(* CODESYS project Tc3_Component.library
   Description: State Model with Observer and Events
   Author: Peter Zerlauth
   Company: Zerlauth
   Version: 0.0.0.1
   Title: Tc3_Component
   DefaultNamespace: Tc3_Component
   Placeholder: Tc3_Component

Project tree, tasks and I/O mapping:
  libraries: Tc2_Standard, * (Beckhoff Automation GmbH); Tc2_System, * (Beckhoff Automation GmbH); Tc2_Utilities, * (Beckhoff Automation GmbH); Tc3_JsonXml, * (Beckhoff Automation GmbH)
  Component/
    Event/
      Observable/
        function block FB_Observable [ST]: FB_exit, M_Attach, M_Clear, M_Detach, M_Find, M_Index, M_Notify, P_Length
        interface I_Observable: M_Attach, M_Detach, P_Length
        interface I_Observer: M_Notify
      data type E_Event
      function block FB_Event [ST]: FB_init, M_Abort, M_AddBOOL, M_AddINT, M_AddREAL, M_AddSTRING, M_AddTIME, M_Arguments, M_Debug, M_Default, M_Error, M_Info, M_Stop, M_Warning, P_History, P_Logger, P_Observer
      interface I_Event: M_Abort, M_AddBOOL, M_AddINT, M_AddREAL, M_AddSTRING, M_AddTIME, M_Debug, M_Error, M_Info, M_Stop, M_Warning, P_History, P_Logger, P_Observer
      data type ST_Event
      data type ST_EventFlags
    Info/
      function block FB_Info [ST]: M_Initialise, P_Class, P_Comment, P_ID, P_Instance, P_Timestamp
      interface I_Info: P_Class, P_Comment, P_ID, P_Instance, P_Timestamp
    Sequence/
      data type E_Sequence
      function block FB_Sequence [ST]: FB_init, M_Await, M_Reset, M_Restore, M_Save, M_Set, P_History, P_Message, P_Number
      interface I_Sequence: M_Await, M_Reset, M_Set, P_History, P_Message, P_Number
      data type ST_Sequence
    data type E_RequestMode
    data type E_RequestState
    data type E_State
    function block FB_Component [ST]: M_RequestMode, M_RequestState, M_Aborted, M_Aborting, M_Completed, M_Completing, M_Execute, M_Held, M_Holding, M_Idle, M_Initialise, M_Paused, M_Pausing, M_Resetting, M_Resuming, M_Running, M_Starting, M_Stopped, M_Stopping, M_Unholding, FB_init, M_Cycle, M_Notify, M_OnMode, M_OnState, P_Event, P_Info, P_Mode, P_Sequence, P_State
    interface I_Component: M_Cycle, M_RequestMode, M_RequestState, P_Event, P_Info, P_Mode, P_State
    interface I_Cycle: M_Cycle
  Function/
    function block FB_Function [ST]
  Images/
    StateModel.svg
    test.jpg
  00000000-0000-0000-0000-000000000000|Images\StateModel.svg
  00000000-0000-0000-0000-000000000000|Images\test.jpg
  Layers/
    Layer/
      function block FB_Layer [ST]: M_Attach, M_Dettach, M_Notify, M_Resetting, M_Starting, P_Delay, P_List, P_Next, P_Timeout
      interface I_Layer: M_Attach, M_Dettach, P_Delay, P_List, P_Next, P_Timeout
    function block FB_Layers [ST]: M_Cycle, P_E0, P_E1, P_On
    interface I_Layers: P_E0, P_E1, P_On
  List/
    function block FB_ListComponent [ST]: FB_exit, M_Add, M_Clear, M_Find, M_Index, M_Remove, P_Length
    function block FB_ListObject [ST]: FB_exit, M_Add, M_Clear, M_Find, M_Index, M_Remove, P_Length
    function block FB_ListString [ST]: FB_exit, M_Add, M_Clear, M_Find, M_Index, M_Remove, P_Length
    interface I_ListBase: M_Clear, P_Length
    interface I_ListComponent: M_Add, M_Find, M_Index, M_Remove
    interface I_ListObject: M_Add, M_Find, M_Index, M_Remove
    interface I_ListString: M_Add, M_Find, M_Index, M_Remove
  Logger/
    function block FB_AbstractLogger [ST]: M_Log, P_LogLevel
    function block FB_GlobalLogger [ST]: M_Find, M_Log
    function block FB_ListObject_1 [ST]: FB_exit, M_Add, M_Clear, M_Find, M_Index, M_Remove, P_Length
    function block FB_Logger [ST]: M_Delete, M_Find, M_Log, M_Reset, P_Events, P_Length
    function block FB_TcLogger [ST]: M_Find, M_Log, M_Reset
    interface I_Logger: M_Log
  Module/
    function block FB_Module [ST]: M_Aborted, M_Completing, M_Cycle, M_Holding, M_Idle, M_Initialise, M_OnMode, M_Pausing, M_Resetting, M_Resuming, M_Running, M_Starting, M_Stopped, M_Unholding, P_Layers
    interface I_Module: P_Layers
  Object/
    function block FB_Object [ST]
    interface I_Object
  Utils/
    Analog/
      function block AnalogInput [ST]: P_ID, P_State, P_Value
      function block AnalogInputREAL [ST]: P_ID, P_State, P_Value
      function block AnalogOutput [ST]: FB_init, P_ID, P_State, P_Value
      interface I_AnalogChannel: P_Value
    Digital/
      function block FB_DigitalInput [ST]: P_ID, P_State, P_Value
      function block FB_DigitalOutput [ST]: P_ID, P_State, P_Value
      interface I_Channel: P_ID, P_State
      interface I_DigitalChannel: P_Value
    File/
      function block FB_File [ST]: M_Append, M_AppendLine, M_Close, M_Create, M_Delete, M_Load, M_Open, M_Read, M_Write, P_Error
      interface I_File: M_Append, M_AppendLine, M_Close, M_Create, M_Delete, M_Load, M_Open, M_Read, M_Write, P_Error
    function block FB_ArrayDint [ST]
    function block FB_Debounce [ST]: P_Value
  Version/
    global variables Global_Version
  global variables Globals
  global variables Parameters
*)

// Component/Event/E_Event
{attribute 'qualified_only'}
{attribute 'strict'}
{attribute 'to_string'}
TYPE E_Event :
(
	Verbose			:= 0,
	Debug			:= 1,
	Information		:= 2,
	Warning			:= 3,
	Error			:= 4
);
END_TYPE

// Component/Event/ST_Event
{attribute 'analysis' := '-33'}
TYPE ST_Event :
	STRUCT
		iSource:		I_Component;
		eEventType:		E_Event;
		nTimestamp:   	ULINT;
		nID:			ULINT;
		sInstance:		STRING(255);
		sClass:			STRING(255);
		sMessage:		STRING(255);
		sDefault:		STRING(255);
		sArguments:		STRING(255);
		stFlags:		ST_EventFlags;
	END_STRUCT
END_TYPE

// Component/Event/ST_EventFlags
{attribute 'analysis' := '-33'}
TYPE ST_EventFlags :
STRUCT
	bActive:		BIT;
	bRemove:		BIT;
END_STRUCT
END_TYPE

// Component/Sequence/E_Sequence
{attribute 'qualified_only'}
{attribute 'strict'}
{attribute 'to_string'}

TYPE E_Sequence :
(
	Manual			:= -32768,
	{attribute 'analysis' := '-27'}
	Start			:= 0,
	Done			:= 32767
);
END_TYPE

// Component/Sequence/ST_Sequence
TYPE ST_Sequence :
STRUCT
	sMessage:				STRING(255);
	nNumber:				INT;
END_STRUCT
END_TYPE

// Component/E_RequestMode
{attribute 'qualified_only'}
{attribute 'strict'}
{attribute 'to_string'}
TYPE E_RequestMode :
(
	{attribute 'hide'}
    Undefined   := 0,
	Automatic   := 1,
    Semiauto    := 2,
	Manual		:= 3
);
END_TYPE

// Component/E_RequestState
{attribute 'qualified_only'}
{attribute 'strict'}
{attribute 'to_string'}

TYPE E_RequestState :
(
	{attribute 'hide'}
    Undefined   := 0,
	{attribute 'analysis' := '-27'}
	Reset       := 1,
	{attribute 'analysis' := '-27'}
    Start       := 2,
    Pause       := 4,	
    Hold      	:= 8,
	Complete	:= 16,	
	Stop		:= 32,
	Abort       := 64
);
END_TYPE

// Component/E_State
{attribute 'qualified_only'}
{attribute 'strict'}
{attribute 'to_string'}
TYPE E_State :
(
	{attribute 'hide'}
	Undefined		:= 0,
	Idle			:= 1,
	
// Start
	Starting		:= 2,
	Execute			:= 3,
	
// Pause
	Pausing			:= 4,
	Paused			:= 5,
	Resuming		:= 6,
	
// Hold
	Holding			:= 7,
	Held			:= 8,
	Unholding		:= 9,
	
// Complete
	Completing		:= 10,
	Completed		:= 11,

// Stop
	Stopping		:= 12,
	Stopped			:= 13,

// Abort	
	Aborting		:= 14,
	Aborted			:= 15,

// Reset
	Resetting		:= 16

);
END_TYPE

// Version/Global_Version
{attribute 'TcGenerated'}
{attribute 'no-analysis'}
{attribute 'linkalways'}
// This function has been automatically generated from the project information.
VAR_GLOBAL CONSTANT
	{attribute 'const_non_replaced'}
	stLibVersion_Tc3_Component : ST_LibVersion := (iMajor := 0, iMinor := 0, iBuild := 0, iRevision := 1, nFlags := 0, sVersion := '0.0.0.1');
END_VAR

// Globals
VAR_GLOBAL
	{IF (defined (release))}
    	{attribute 'hide'}
	{END_IF}
	fbLogger:			FB_GlobalLogger;		// Global Logger, as default without module
	{attribute 'analysis' := '-33'}
	bSimulation:		BOOL;
END_VAR

// Parameters
{attribute 'qualified_only'}
VAR_GLOBAL CONSTANT
	{attribute 'analysis' := '-33'}
	nSequence:						UINT:= 9;		// Maximum of Sequence history
	{attribute 'analysis' := '-33'}
	nList:							UINT:= 46;		// Maximum of displayed items in list
END_VAR

// Component/Event/Observable/FB_Observable
{attribute 'no_explicit_call'} 
FUNCTION_BLOCK PUBLIC FB_Observable IMPLEMENTS I_Observable
VAR_INPUT
	iParent:		I_Component;	
END_VAR
VAR
	pList: 			POINTER TO I_Component;
    {attribute 'hide'}
	nLength:		DINT;
	{IF (defined (release))}
    	{attribute 'hide'}
	{END_IF}
	aList:			POINTER TO POINTER TO ARRAY [0..100] OF I_Component:=ADR(pList);
END_VAR

// https://github.com/PeterZerlauth/Tc3_Component

METHOD FB_exit : BOOL
VAR_INPUT
	bInCopyCode : BOOL; // if TRUE, the exit method is called for exiting an instance that is copied afterwards (online change).
END_VAR
M_Clear();
END_METHOD

METHOD M_Attach : BOOL
VAR_INPUT
	Object: 	I_Component;
END_VAR
VAR
	pOldList: 	POINTER TO I_Component;
END_VAR
IF Object <> 0 THEN
	// First Item
	IF pList = 0 THEN
		nLength:= nLength + 1;
		pList:= __NEW(POINTER TO I_Component,DINT_TO_UDINT(nLength));
	ELSE
		// Item already in List
		IF M_Find(Object) = -1 THEN
			// backup 
			pOldList:= pList;
			// new Length
			nLength:= nLength + 1;
			// new pointer
			pList:= __NEW(POINTER TO I_Component,DINT_TO_UDINT(nLength));
			// restore
			Memcpy(pList,pOldList, SIZEOF(POINTER TO I_Component)*DINT_TO_UDINT(nLength -1));
			// delete old
			__DELETE(pOldList);
		ELSE
			M_Attach:= FALSE;	
			RETURN;
		END_IF
	END_IF
	IF pList = 0 THEN
		RETURN;
	END_IF
	// add new Object
	pList[nLength-1]:= Object;
	M_Attach:= TRUE;
ELSE
	M_Attach:= FALSE;	
END_IF
END_METHOD

METHOD M_Clear
IF pList <> 0 THEN
	nLength:= 0;
	__DELETE(pList);
END_IF
END_METHOD

METHOD M_Detach : BOOL
VAR_INPUT
	Object: 	I_Component;
END_VAR
VAR
	pOldList:			POINTER TO I_Component;
	nPosition: 			DINT;
END_VAR
IF Object <> 0 THEN
	// First Item
	IF nLength >= 0 THEN
		// Item already in List
		nPosition:= M_Find(Object);
		IF nPosition <> -1 THEN
			// backup 
			pOldList:= pList;
			// new Length
			nLength:= nLength -1;
			// new pointer
			pList:= __NEW(POINTER TO I_Component,DINT_TO_UDINT(nLength));
			// restore lower part
			Memcpy(pList,pOldList, SIZEOF(POINTER TO I_Component) * DINT_TO_UDINT(nPosition));
			//pList[nPosition]:= iObject;
			Memcpy(pList + (SIZEOF(POINTER TO I_Component)*nPosition),pOldList + (SIZEOF(POINTER TO I_Component)*(nPosition + 1)), SIZEOF(POINTER TO I_Component) * DINT_TO_UDINT(nLength - nPosition));
			// delete old
			__DELETE(pOldList);
		ELSE
			M_Detach:= FALSE;	
			RETURN;
		END_IF
	ELSE
		M_Detach:= FALSE;	
		RETURN;
	END_IF
	M_Detach:= TRUE;
ELSE
	M_Detach:= FALSE;	
END_IF
END_METHOD

METHOD M_Find : DINT
VAR_INPUT
	Object: 	I_Component;
END_VAR
VAR
	nIndex: 	UINT;
END_VAR
// Object already in List
M_Find := -1;
WHILE nIndex < nLength DO
    IF (pList[nIndex] = Object) THEN
        M_Find := nIndex;
        RETURN;
    END_IF
	nIndex := nIndex + 1;
END_WHILE
END_METHOD

METHOD M_Index : I_Observer
VAR_INPUT
	Index: 	DINT;
END_VAR
IF Index <= nLength THEN
	M_Index:= pList[Index];
END_IF
END_METHOD

METHOD M_Notify
VAR_INPUT
	iSender:		I_Component;
	eRequest:		E_RequestState;
END_VAR

VAR
	nIndex: 		DINT;
END_VAR
// Prevent Infinite loop from callbacks
WHILE nIndex < nLength DO
	IF pList[nIndex] <> iSender THEN
		pList[nIndex].M_Notify(iParent, eRequest);		
	END_IF
	nIndex:= nIndex + 1; 
END_WHILE
END_METHOD

{attribute 'OPC.UA.DA.Property' := '1'}
{attribute 'monitoring' := 'call'}
PROPERTY P_Length : DINT
GET
P_Length:= nLength;
END_GET
END_PROPERTY

END_FUNCTION_BLOCK

// Component/Event/Observable/I_Observable
INTERFACE I_Observable EXTENDS I_Observer

METHOD PUBLIC M_Attach : BOOL
VAR_INPUT
	Object: 	I_Component;
END_VAR
END_METHOD

METHOD PUBLIC M_Detach : BOOL
VAR_INPUT
	Object: 	I_Component;
END_VAR
END_METHOD

{attribute 'OPC.UA.DA.Property' := '1'}
{attribute 'monitoring' := 'call'}
PROPERTY P_Length : DINT
GET
END_GET
END_PROPERTY

END_INTERFACE

// Component/Event/Observable/I_Observer
INTERFACE I_Observer EXTENDS I_Object

METHOD PUBLIC M_Notify
VAR_INPUT
	iSender:		I_Component;
	eRequest:		E_RequestState;
END_VAR
END_METHOD

END_INTERFACE

// Object/I_Object
INTERFACE I_Object EXTENDS __SYSTEM.IQueryInterface

END_INTERFACE

// Component/I_Component
INTERFACE I_Component EXTENDS I_Observer, I_Cycle

METHOD PUBLIC M_Cycle
VAR_INPUT
END_VAR
END_METHOD

METHOD PUBLIC M_RequestMode : BOOL
VAR_INPUT
	eMode:		E_RequestMode;
END_VAR
END_METHOD

METHOD PUBLIC M_RequestState : BOOL
VAR_INPUT
	eRequest:	E_RequestState;
END_VAR
END_METHOD

PROPERTY PUBLIC P_Event : I_Event
GET
END_GET
END_PROPERTY

{attribute 'OPC.UA.DA.Property' := '1'}
{attribute 'monitoring' := 'call'}
PROPERTY PUBLIC P_Info : I_Info
GET
END_GET
END_PROPERTY

{attribute 'OPC.UA.DA.Property' := '1'}
{attribute 'monitoring' := 'call'}
PROPERTY PUBLIC P_Mode : E_RequestMode
GET
END_GET
END_PROPERTY

{attribute 'OPC.UA.DA.Property' := '1'}
{attribute 'monitoring' := 'call'}
PROPERTY PUBLIC P_State : E_State
GET
END_GET
END_PROPERTY

END_INTERFACE

// Component/I_Cycle
INTERFACE I_Cycle EXTENDS I_Object

METHOD PUBLIC M_Cycle
VAR_INPUT
END_VAR
END_METHOD

END_INTERFACE

// Component/Event/I_Event
INTERFACE I_Event EXTENDS I_Object

METHOD PUBLIC M_Abort
VAR_INPUT
	sMessage:				STRING(255);
	nID:					ULINT;
END_VAR
END_METHOD

METHOD PUBLIC M_AddBOOL : I_Event
VAR_INPUT
	Value: 	BOOL;
END_VAR
END_METHOD

METHOD PUBLIC M_AddINT : I_Event
VAR_INPUT
	Value: 	LINT;
END_VAR
END_METHOD

METHOD PUBLIC M_AddREAL : I_Event
VAR_INPUT
	Value: 	Lreal;
	Decimals: INT;
END_VAR
END_METHOD

METHOD PUBLIC M_AddSTRING : I_Event
VAR_INPUT
	Value: STRING(255);
END_VAR
END_METHOD

METHOD PUBLIC M_AddTIME : I_Event
VAR_INPUT
	Value: 	TIME;
END_VAR
END_METHOD

METHOD PUBLIC M_Debug
VAR_INPUT
	sMessage:				STRING(255);
END_VAR
END_METHOD

METHOD PUBLIC M_Error
VAR_INPUT
	sMessage:				STRING(255);
	nID:					ULINT;
END_VAR
END_METHOD

METHOD PUBLIC M_Info
VAR_INPUT
	sMessage:				STRING(255);
	nID:					ULINT;
END_VAR
END_METHOD

METHOD PUBLIC M_Stop
VAR_INPUT
	sMessage:				STRING(255);
	nID:					ULINT;
END_VAR
END_METHOD

METHOD PUBLIC M_Warning
VAR_INPUT
	sMessage:				STRING(255);
	nID:					ULINT;
END_VAR
END_METHOD

{attribute 'OPC.UA.DA.Property' := '1'}
{attribute 'monitoring' := 'call'}
{attribute 'suppress_wrn_C0410'}
PROPERTY PUBLIC P_History : REFERENCE TO ARRAY [0..5] OF ST_Event;
GET
END_GET
SET
END_SET
END_PROPERTY

PROPERTY PUBLIC P_Logger : I_Logger
GET
END_GET
SET
END_SET
END_PROPERTY

PROPERTY PUBLIC P_Observer : I_Observable
GET
END_GET
END_PROPERTY

END_INTERFACE

// Logger/I_Logger
INTERFACE I_Logger EXTENDS I_Object

METHOD PUBLIC M_Log
VAR_INPUT
	{attribute 'analysis' := '-33'}
	stEvent	: ST_Event;
END_VAR
END_METHOD

END_INTERFACE

// Component/Info/I_Info
INTERFACE I_Info EXTENDS I_Object

{attribute 'OPC.UA.DA.Property' := '1'}
{attribute 'monitoring' := 'call'}
PROPERTY PUBLIC P_Class : STRING(255)
GET
END_GET
END_PROPERTY

{attribute 'OPC.UA.DA.Property' := '1'}
{attribute 'monitoring' := 'call'}
PROPERTY PUBLIC P_Comment : STRING(255)
GET
END_GET
END_PROPERTY

{attribute 'OPC.UA.DA.Property' := '1'}
{attribute 'monitoring' := 'call'}
PROPERTY PUBLIC P_ID : STRING(25)
GET
END_GET
SET
END_SET
END_PROPERTY

{attribute 'OPC.UA.DA.Property' := '1'}
{attribute 'monitoring' := 'call'}
PROPERTY PUBLIC P_Instance : STRING(255)
GET
END_GET
END_PROPERTY

{attribute 'OPC.UA.DA.Property' := '1'}
{attribute 'monitoring' := 'call'}
PROPERTY PUBLIC P_Timestamp : ULINT
GET
END_GET
END_PROPERTY

END_INTERFACE

// Component/Event/FB_Event
FUNCTION_BLOCK FB_Event IMPLEMENTS I_Event
VAR_INPUT
	fbObserver:			FB_Observable;				// Observer
END_VAR
VAR_OUTPUT
END_VAR
VAR
	iLogger:			I_Logger;
	iParent:			I_Component;				// Parent component
    {attribute 'hide'}
	fbList:				FB_ListString;				// contains a list with string values

	stEvent:			ST_Event;					// Event
    {attribute 'hide'}
	aHistory:			ARRAY [0..5] OF ST_Event;	// History of events
END_VAR

// https://github.com/PeterZerlauth/Tc3_Component

METHOD FB_init : BOOL
VAR_INPUT
	bInitRetains : BOOL; // if TRUE, the retain variables are initialized (warm start / cold start)
	bInCopyCode : BOOL;  // if TRUE, the instance afterwards gets moved into the copy code (online change)
	iParent:			I_Component;
END_VAR
THIS^.iParent:= iParent;
fbObserver.iParent:= iParent;
END_METHOD

METHOD PUBLIC M_Abort
VAR_INPUT
	sMessage:				STRING(255);
	nID:					ULINT;
END_VAR
stEvent.sMessage:= sMessage;
stEvent.iSource:= iParent;
stEvent.sInstance:= iParent.P_Info.P_Instance;
stEvent.sClass:= iParent.P_Info.P_Class;
stEvent.eEventType:= E_Event.Error;
stEvent.nTimestamp:= F_GetSystemTime();
stEvent.nID:= nID;
stEvent.sDefault:= M_Default(sMessage);
stEvent.sArguments:= M_Arguments();
stEvent.stFlags.bActive:= TRUE;
stEvent.stFlags.bRemove:= FALSE;

IF iLogger = 0 THEN
	fbLogger.M_Log(stEvent);
ELSE
	iLogger.M_Log(stEvent);
END_IF

iParent.M_RequestState(E_RequestState.Abort);

fbObserver.M_Notify(iParent, E_RequestState.Abort);

IF aHistory[0].sMessage <> stEvent.sMessage THEN
	MemCpy(ADR(aHistory[1]), ADR(aHistory[0]), SIZEOF(ST_Event) * 5);
	aHistory[0]:= stEvent;
END_IF
END_METHOD

METHOD PUBLIC M_AddBOOL : I_Event
VAR_INPUT
	Value: 	bool;
END_VAR
fbList.M_Add(BOOL_TO_STRING(Value));
M_AddBOOL:= THIS^;
END_METHOD

METHOD PUBLIC M_AddINT : I_Event
VAR_INPUT
	Value: 	LINT;
END_VAR
fbList.M_Add(LINT_TO_STRING(Value));
M_AddINT:= THIS^;
END_METHOD

METHOD PUBLIC M_AddREAL : I_Event
VAR_INPUT
	Value: 	Lreal;
	Decimals: INT;
END_VAR
fbList.M_Add(LREAL_TO_FMTSTR(Value, Decimals, TRUE));
M_AddREAL:= THIS^;
END_METHOD

METHOD PUBLIC M_AddSTRING : I_Event
VAR_INPUT
	Value: STRING(255);
END_VAR
fbList.M_Add(Value);
M_AddSTRING:= THIS^;
END_METHOD

METHOD PUBLIC M_AddTIME : I_Event
VAR_INPUT
	Value: 	TIME;
END_VAR
fbList.M_Add(TIME_TO_STRING(Value));
M_AddTIME:= THIS^;
END_METHOD

METHOD INTERNAL M_Arguments : STRING(255)
VAR_INPUT
END_VAR
VAR
	nIndex:			INT;
END_VAR
WHILE nIndex < fbList. P_Length DO
	M_Arguments:= Concat(Concat(M_Arguments, fbList.M_Index(nIndex)), '$N');
	nIndex:= nIndex + 1;
END_WHILE

fbList.M_Clear();
END_METHOD

METHOD PUBLIC M_Debug
VAR_INPUT
	sMessage:				STRING(255);
END_VAR
stEvent.sMessage:= sMessage;
stEvent.iSource:= iParent;
stEvent.sInstance:= iParent.P_Info.P_Instance;
stEvent.sClass:= iParent.P_Info.P_Class;
stEvent.eEventType:= E_Event.Debug;
stEvent.nTimestamp:= F_GetSystemTime();
stEvent.nID:= 0;
stEvent.sDefault:= M_Default(sMessage);
stEvent.sArguments:= M_Arguments();
stEvent.stFlags.bActive:= TRUE;
stEvent.stFlags.bRemove:= TRUE;

IF iLogger = 0 THEN
	fbLogger.M_Log(stEvent);
ELSE
	iLogger.M_Log(stEvent);
END_IF

IF aHistory[0].sMessage <> stEvent.sMessage THEN
	MemCpy(ADR(aHistory[1]), ADR(aHistory[0]), SIZEOF(ST_Event) * 5);
	aHistory[0]:= stEvent;
END_IF
END_METHOD

METHOD INTERNAL M_Default : STRING(255)
VAR_INPUT
	sMessage:		STRING(255);
END_VAR
VAR
	nIndex:		   	DINT;
	nPosition: 		INT;
END_VAR
nPosition:= Find(sMessage, '%s');
WHILE nPosition <> 0 DO
	sMessage:= Replace(sMessage, fbList.M_Index(nIndex), 2, nPosition);
	nPosition:= Find(sMessage, '%s');
	nIndex:= nIndex + 1;
END_WHILE
M_Default:= sMessage;
END_METHOD

METHOD PUBLIC M_Error
VAR_INPUT
	sMessage:				STRING(255);
	nID:					ULINT;
END_VAR
stEvent.sMessage:= sMessage;
stEvent.iSource:= iParent;
stEvent.sInstance:= iParent.P_Info.P_Instance;
stEvent.sClass:= iParent.P_Info.P_Class;
stEvent.eEventType:= E_Event.Error;
stEvent.nTimestamp:= F_GetSystemTime();
stEvent.nID:= nID;
stEvent.sDefault:= M_Default(sMessage);
stEvent.sArguments:= M_Arguments();
stEvent.stFlags.bActive:= TRUE;
stEvent.stFlags.bRemove:= TRUE;

IF iLogger = 0 THEN
	fbLogger.M_Log(stEvent);
ELSE
	iLogger.M_Log(stEvent);
END_IF

IF aHistory[0].sMessage <> stEvent.sMessage THEN
	MemCpy(ADR(aHistory[1]), ADR(aHistory[0]), SIZEOF(ST_Event) * 5);
	aHistory[0]:= stEvent;
END_IF
END_METHOD

METHOD PUBLIC M_Info
VAR_INPUT
	sMessage:				STRING(255);
	nID:					ULINT;
END_VAR
stEvent.sMessage:= sMessage;
stEvent.iSource:= iParent;
stEvent.sInstance:= iParent.P_Info.P_Instance;
stEvent.sClass:= iParent.P_Info.P_Class;
stEvent.eEventType:= E_Event.Information;
stEvent.nTimestamp:= F_GetSystemTime();
stEvent.nID:= nID;
stEvent.sDefault:= M_Default(sMessage);
stEvent.sArguments:= M_Arguments();
stEvent.stFlags.bActive:= TRUE;
stEvent.stFlags.bRemove:= TRUE;

IF iLogger = 0 THEN
	fbLogger.M_Log(stEvent);
ELSE
	iLogger.M_Log(stEvent);
END_IF

IF aHistory[0].sMessage <> stEvent.sMessage THEN
	MemCpy(ADR(aHistory[1]), ADR(aHistory[0]), SIZEOF(ST_Event) * 5);
	aHistory[0]:= stEvent;
END_IF
END_METHOD

METHOD PUBLIC M_Stop
VAR_INPUT
	sMessage:				STRING(255);
	nID:					ULINT;
END_VAR
stEvent.sMessage:= sMessage;
stEvent.iSource:= iParent;
stEvent.sInstance:= iParent.P_Info.P_Instance;
stEvent.sClass:= iParent.P_Info.P_Class;
stEvent.eEventType:= E_Event.Error;
stEvent.nTimestamp:= F_GetSystemTime();
stEvent.nID:= nID;
stEvent.sDefault:= M_Default(sMessage);
stEvent.sArguments:= M_Arguments();
stEvent.stFlags.bActive:= TRUE;
stEvent.stFlags.bRemove:= FALSE;

IF iLogger = 0 THEN
	fbLogger.M_Log(stEvent);
ELSE
	iLogger.M_Log(stEvent);
END_IF

iParent.M_RequestState(E_RequestState.Stop);

fbObserver.M_Notify(iParent, E_RequestState.Abort);

IF aHistory[0].sMessage <> stEvent.sMessage THEN
	MemCpy(ADR(aHistory[1]), ADR(aHistory[0]), SIZEOF(ST_Event) * 5);
	aHistory[0]:= stEvent;
END_IF
END_METHOD

METHOD PUBLIC M_Warning
VAR_INPUT
	sMessage:				STRING(255);
	nID:					ULINT;
END_VAR
stEvent.sMessage:= sMessage;
stEvent.iSource:= iParent;
stEvent.sInstance:= iParent.P_Info.P_Instance;
stEvent.sClass:= iParent.P_Info.P_Class;
stEvent.eEventType:= E_Event.Warning;
stEvent.nTimestamp:= F_GetSystemTime();
stEvent.nID:= nID;
stEvent.sDefault:= M_Default(sMessage);
stEvent.sArguments:= M_Arguments();
stEvent.stFlags.bActive:= TRUE;
stEvent.stFlags.bRemove:= TRUE;

IF iLogger = 0 THEN
	fbLogger.M_Log(stEvent);
ELSE
	iLogger.M_Log(stEvent);
END_IF

IF aHistory[0].sMessage <> stEvent.sMessage THEN
	MemCpy(ADR(aHistory[1]), ADR(aHistory[0]), SIZEOF(ST_Event) * 5);
	aHistory[0]:= stEvent;
END_IF
END_METHOD

{attribute 'OPC.UA.DA.Property' := '1'}
{attribute 'monitoring' := 'call'}
{attribute 'suppress_wrn_C0410'}
PROPERTY PUBLIC P_History : REFERENCE TO ARRAY [0..5] OF ST_Event;
GET
P_History REF= aHistory;
END_GET
SET
P_History REF= aHistory;
END_SET
END_PROPERTY

PROPERTY P_Logger : I_Logger
GET
P_Logger:= iLogger;
END_GET
SET
iLogger:= P_Logger;
END_SET
END_PROPERTY

PROPERTY PUBLIC P_Observer : I_Observable
GET
P_Observer:= fbObserver;
END_GET
END_PROPERTY

END_FUNCTION_BLOCK

// List/FB_ListString
{attribute 'no_explicit_call' := 'do not call this POU directly'} 
FUNCTION_BLOCK FB_ListString IMPLEMENTS I_ListString
VAR
	pList: 			POINTER TO STRING(255);
	nLength:		DINT;
	{IF (defined (release))}
    	{attribute 'hide'}
	{END_IF}
	aList:			POINTER TO POINTER TO ARRAY [0..Parameters.nList] OF STRING(255):=ADR(pList);
END_VAR
(*!<example> This sample shows how to use the function block</c>.

The following code can be used to add string variable
<code>fbList.M_Add('string item');</code>


</example>*)

// https://github.com/PeterZerlauth/Tc3_Component

METHOD FB_exit : BOOL
VAR_INPUT
	bInCopyCode : BOOL; // if TRUE, the exit method is called for exiting an instance that is copied afterwards (online change).
END_VAR
M_Clear();
END_METHOD

METHOD PUBLIC M_Add : BOOL
VAR_INPUT
	Object: 	STRING(255);
END_VAR
VAR
	pOldList: 	POINTER TO STRING(255);
END_VAR
IF Object <> '' THEN
	// First Item
	IF pList = 0 THEN
		nLength:= nLength + 1;
		pList:= __NEW(STRING(255),DINT_TO_UDINT(nLength));
	ELSE
		// Item already in List
		IF M_Find(Object) = -1 THEN
			// backup 
			pOldList:= pList;
			// new Length
			nLength:= nLength + 1;
			// new pointer
			pList:= __NEW(STRING(255),DINT_TO_UDINT(nLength));
			// restore
			Memcpy(pList,pOldList, SIZEOF(STRING(255))*DINT_TO_UDINT(nLength -1));
			// delete old
			__DELETE(pOldList);
		ELSE
			M_Add:= FALSE;	
			RETURN;
		END_IF
	END_IF
	IF pList = 0 THEN
		RETURN;
	END_IF
	// add new Object
	pList[nLength-1]:= Object;
	M_Add:= TRUE;
ELSE
	M_Add:= FALSE;	
END_IF
END_METHOD

METHOD PUBLIC M_Clear : BOOL
IF pList <> 0 THEN
	nLength:= 0;
	__DELETE(pList);
END_IF
M_Clear:= True;
END_METHOD

METHOD PUBLIC M_Find : DINT
VAR_INPUT
	Object: 	STRING(255);
END_VAR
VAR
	nIndex: 	UINT;
END_VAR
// Object already in List
M_Find := -1;
WHILE nIndex < nLength DO
    IF (pList[nIndex] = Object) THEN
        M_Find := nIndex;
        RETURN;
    END_IF
	nIndex := nIndex + 1;
END_WHILE
END_METHOD

METHOD PUBLIC M_Index : STRING(255)
VAR_INPUT
	Index: 	DINT;
END_VAR
IF Index <= nLength THEN
	M_Index:= pList[Index];
ELSE
	M_Index:= '';
END_IF
END_METHOD

METHOD PUBLIC M_Remove : BOOL
VAR_INPUT
	Object: 	STRING(255);
END_VAR
VAR
	pOldList:			POINTER TO STRING(255);
	nPosition: 			DINT;
END_VAR
IF Object <> '' THEN
	// First Item
	IF nLength >= 0 THEN
		// Item already in List
		nPosition:= M_Find(Object);
		IF nPosition <> -1 THEN
			// backup 
			pOldList:= pList;
			// new Length
			nLength:= nLength -1;
			// new pointer
			pList:= __NEW(POINTER TO I_Object,DINT_TO_UDINT(nLength));
			// restore lower part
			Memcpy(pList,pOldList, SIZEOF(STRING(255)) * DINT_TO_UDINT(nPosition));
			//pList[nPosition]:= iObject;
			Memcpy(pList + (SIZEOF(STRING(255))*nPosition),pOldList + (SIZEOF(STRING(255))*(nPosition + 1)), SIZEOF(STRING(255)) * DINT_TO_UDINT(nLength - nPosition));
			// delete old
			__DELETE(pOldList);
		ELSE
			M_Remove:= FALSE;	
			RETURN;
		END_IF
	ELSE
		M_Remove:= FALSE;	
		RETURN;
	END_IF
	M_Remove:= TRUE;
ELSE
	M_Remove:= FALSE;	
END_IF
END_METHOD

{attribute 'OPC.UA.DA.Property' := '1'}
{attribute 'monitoring' := 'call'}
PROPERTY PUBLIC P_Length : DINT
GET
P_Length:= nLength;
END_GET
END_PROPERTY

END_FUNCTION_BLOCK

// List/I_ListString
INTERFACE I_ListString EXTENDS I_ListBase

METHOD PUBLIC M_Add : BOOL
VAR_INPUT
	Object: 	STRING(255);
END_VAR
END_METHOD

METHOD PUBLIC M_Find : DINT
VAR_INPUT
	Object: 	STRING(255);
END_VAR
END_METHOD

METHOD PUBLIC M_Index : STRING(255)
VAR_INPUT
	Index: 	DINT;
END_VAR
END_METHOD

METHOD PUBLIC M_Remove : BOOL
VAR_INPUT
	Object: 	STRING(255);
END_VAR
END_METHOD

END_INTERFACE

// List/I_ListBase
INTERFACE I_ListBase EXTENDS I_Object

METHOD PUBLIC M_Clear : BOOL
END_METHOD

{attribute 'OPC.UA.DA.Property' := '1'}
{attribute 'monitoring' := 'call'}
PROPERTY public P_Length : DINT
GET
END_GET
END_PROPERTY

END_INTERFACE

// Component/Info/FB_Info
{attribute 'reflection'} 
FUNCTION_BLOCK PUBLIC FB_Info IMPLEMENTS I_Info
VAR_INPUT
END_VAR
VAR_OUTPUT
END_VAR
VAR
	sIdentifier:						STRING(25):= 'Identifier';				// Identifier
	{attribute 'instance-path'} 
    {attribute 'noinit'}
    sInstancePath:				STRING(255);									// Instance-Path
	fbReadSymInfo: 				PLC_ReadSymInfoByNameEx;						// Read symbol infos
END_VAR
VAR_STAT
	nCycle: 					UDINT;
	nTimestamp: 				ULINT;
END_VAR

// https://github.com/PeterZerlauth/Tc3_Component

// Update once for all function blocks
IF nCycle <> TwinCAT_SystemInfoVarList._TaskInfo[GETCURTASKINDEXEX()].CycleCount THEN
	nCycle:= TwinCAT_SystemInfoVarList._TaskInfo[GETCURTASKINDEXEX()].CycleCount;
	nTimestamp:= F_GetSystemTime();
END_IF

// Read symbol information
fbReadSymInfo();
IF NOT fbReadSymInfo.START THEN
	M_Initialise();
	fbReadSymInfo.PORT:= TwinCAT_SystemInfoVarList._AppInfo.AdsPort;
	fbReadSymInfo.START:= TRUE;
END_IF

METHOD PROTECTED M_Initialise
VAR_INPUT
END_VAR
VAR
    sName:				STRING(255);
    nPosition:			INT;
END_VAR
sName := CONCAT(TwinCAT_SystemInfoVarList._AppInfo.ProjectName, '.');

nPosition := FIND(sInstancePath, sName);
IF nPosition > 0 THEN
    fbReadSymInfo.SYMNAME:= DELETE(sInstancePath, nPosition-1 + LEN(sName), 1);
END_IF

nPosition := FIND(fbReadSymInfo.SYMNAME, sName);

IF nPosition > 0 THEN
    fbReadSymInfo.SYMNAME:= DELETE(fbReadSymInfo.SYMNAME, nPosition - 1 + LEN(sName), 1);
END_IF

fbReadSymInfo.SYMNAME:= Left(fbReadSymInfo.SYMNAME, LEN(fbReadSymInfo.SYMNAME) - 7);
END_METHOD

{attribute 'OPC.UA.DA.Property' := '1'}
{attribute 'monitoring' := 'call'}
PROPERTY PUBLIC P_Class : STRING(255)
GET
{attribute 'OPC.UA.DA.Property' := '1'}
{attribute 'monitoring' := 'call'}
VAR
END_VAR
P_Class:= fbReadSymInfo.SYMINFO.symDataType;
END_GET
END_PROPERTY

{attribute 'OPC.UA.DA.Property' := '1'}
{attribute 'monitoring' := 'call'}
PROPERTY PUBLIC P_Comment : STRING(255)
GET
P_Comment:= fbReadSymInfo.SYMINFO.symComment;
END_GET
END_PROPERTY

{attribute 'OPC.UA.DA.Property' := '1'}
{attribute 'monitoring' := 'call'}
PROPERTY PUBLIC P_ID : STRING(25)
GET
P_ID:= sIdentifier;
END_GET
SET
PUBLIC 
VAR
END_VAR
sIdentifier:= P_ID;
END_SET
END_PROPERTY

{attribute 'OPC.UA.DA.Property' := '1'}
{attribute 'monitoring' := 'call'}
PROPERTY PUBLIC P_Instance : STRING(255)
GET
P_Instance:= fbReadSymInfo.SYMNAME;
END_GET
END_PROPERTY

{attribute 'OPC.UA.DA.Property' := '1'}
{attribute 'monitoring' := 'call'}
PROPERTY PUBLIC P_Timestamp : ULINT
GET
P_Timestamp:= nTimestamp;
END_GET
END_PROPERTY

END_FUNCTION_BLOCK

// Component/Sequence/FB_Sequence
FUNCTION_BLOCK FB_Sequence IMPLEMENTS I_Sequence
VAR
	iParent:			I_Component;
	stActual:			ST_Sequence;
	stRestore:			ST_Sequence;
	aHistory:			ARRAY [0..Parameters.nSequence] OF ST_Sequence;
	fbTimeout:			TON;
	fbDelay: 			TON;
END_VAR

// https://github.com/PeterZerlauth/Tc3_Component
fbTimeout();
fbTimeout.IN:= FALSE;

fbDelay();
fbDelay.IN:= FALSE;

METHOD FB_init : BOOL
VAR_INPUT
	bInitRetains : BOOL; // if TRUE, the retain variables are initialized (warm start / cold start)
	bInCopyCode : BOOL;  // if TRUE, the instance afterwards gets moved into the copy code (online change)
	iParent:			I_Component;
END_VAR
THIS^.iParent:= iParent;
END_METHOD

METHOD PUBLIC M_Await 
VAR_INPUT
	sMessage:				STRING(255);		
	tTimeout:				TIME;
	tDelay:					TIME;	
	bPause:					BOOL;
	bReturn:				BOOL;
	nNumber:				INT;
END_VAR
IF bReturn THEN
	IF tDelay <> T#0S THEN
		fbDelay.PT:= tDelay;
		fbDelay.IN:= TRUE;
		IF fbDelay.Q THEN
			stActual.sMessage:= sMessage;;
			MemCpy(ADR(aHistory[1]), ADR(aHistory[0]), SIZEOF(ST_Sequence) * Parameters.nSequence);
			aHistory[0]:= stActual;
			stActual.nNumber:= nNumber;
			fbDelay(IN:= FALSE);
			IF bPause THEN
				IF iParent.P_Mode = E_RequestMode.Semiauto THEN
					iParent.M_RequestState(E_RequestState.Pause);		
				END_IF
			END_IF
		END_IF
	ELSE
		stActual.sMessage:= sMessage;
		MemCpy(ADR(aHistory[1]), ADR(aHistory[0]), SIZEOF(ST_Sequence) * Parameters.nSequence);
		aHistory[0]:= stActual;
		stActual.nNumber:= nNumber;
		fbTimeout(IN:= FALSE);
		IF bPause THEN
			IF iParent.P_Mode = E_RequestMode.Semiauto THEN
				iParent.M_RequestState(E_RequestState.Pause);		
			END_IF
		END_IF	
	END_IF		
ELSE
	IF tTimeout <> T#0S THEN
		fbTimeout.PT:= tTimeout;
		fbTimeout.IN:= TRUE;
		IF fbTimeout.Q THEN
			iParent.P_Event.M_AddINT(stActual.nNumber);
			iParent.P_Event.M_Stop('Timeout in sequence number %s', 1);
		END_IF
	END_IF
END_IF
END_METHOD

METHOD PUBLIC M_Reset
stActual.nNumber:= E_Sequence.Start;
stActual.sMessage:= 'E_Sequence.Start';
fbDelay(IN:= FALSE);
fbTimeout(IN:= FALSE);
END_METHOD

METHOD PUBLIC M_Restore
stActual:= stRestore;
END_METHOD

METHOD PUBLIC M_Save
VAR_INPUT
END_VAR
stRestore:= stActual;
END_METHOD

METHOD PUBLIC M_Set
VAR_INPUT
	nNumber:				INT;
END_VAR
stActual.nNumber:= nNumber;
stActual.sMessage:= 'M_Set';
MemCpy(ADR(aHistory[1]), ADR(aHistory[0]), SIZEOF(ST_Sequence) * Parameters.nSequence);
aHistory[0]:= stActual;
fbDelay(IN:= FALSE);
fbTimeout(IN:= FALSE);
END_METHOD

{attribute 'OPC.UA.DA.Property' := '1'}
{attribute 'monitoring' := 'call'}
{attribute 'suppress_wrn_C0410'}
PROPERTY PUBLIC P_History : REFERENCE TO ARRAY [0..Parameters.nSequence] OF ST_Sequence;
GET
P_History REF= aHistory;
END_GET
SET
P_History REF= aHistory;
END_SET
END_PROPERTY

{attribute 'OPC.UA.DA.Property' := '1'}
{attribute 'monitoring' := 'call'}
PROPERTY PUBLIC P_Message : STRING(255)
GET
P_Message:= stActual.sMessage;
END_GET
END_PROPERTY

{attribute 'OPC.UA.DA.Property' := '1'}
{attribute 'monitoring' := 'call'}
PROPERTY PUBLIC P_Number : INT
GET
P_Number:= stActual.nNumber;
END_GET
END_PROPERTY

END_FUNCTION_BLOCK

// Component/Sequence/I_Sequence
INTERFACE I_Sequence EXTENDS I_Object

METHOD PUBLIC M_Await 
VAR_INPUT
	sMessage:				STRING(255);
	tTimeout:				TIME;
	tDelay:					TIME;	
	bPause:					BOOL;
	bReturn:				BOOL;
	nNumber:				INT;
END_VAR
END_METHOD

METHOD PUBLIC M_Reset
END_METHOD

METHOD PUBLIC M_Set
VAR_INPUT
	nNumber:				INT;
END_VAR
END_METHOD

{attribute 'OPC.UA.DA.Property' := '1'}
{attribute 'monitoring' := 'call'}
{attribute 'suppress_wrn_C0410'}
PROPERTY PUBLIC P_History : REFERENCE TO ARRAY [0..Parameters.nSequence] OF ST_Sequence;
GET
END_GET
SET
END_SET
END_PROPERTY

{attribute 'OPC.UA.DA.Property' := '1'}
{attribute 'monitoring' := 'call'}
PROPERTY PUBLIC P_Message : STRING(255)
GET
END_GET
END_PROPERTY

{attribute 'OPC.UA.DA.Property' := '1'}
{attribute 'monitoring' := 'call'}
PROPERTY PUBLIC P_Number : int
GET
END_GET
END_PROPERTY

END_INTERFACE

// Component/FB_Component
{attribute 'no_explicit_call' := 'do not call this POU directly'} 
FUNCTION_BLOCK FB_Component EXTENDS FB_Object IMPLEMENTS I_Component, I_Observer
VAR_INPUT
END_VAR
VAR_OUTPUT
END_VAR
VAR
    {attribute 'hide'}
	fbInfo:							FB_Info;					// Info about function block
	fbEvent:						FB_Event(THIS^);			// Event creator
	fbSequence:						FB_Sequence(THIS^);			// Sequence (abort = reset)
	{attribute 'OPC.UA.DA' := '1'}
	{attribute 'OPC.UA.DA.Access' := '1'}
	eStateRequest:					E_RequestState;					// State command
    {attribute 'hide'}
	eState:							E_State;					// Current state
    {attribute 'hide'}
	eStatePrevious:					E_State;					// Previous state
	{attribute 'OPC.UA.DA' := '1'}
	{attribute 'OPC.UA.DA.Access' := '1'}
	eModeRequest:					E_RequestMode;						// Requested mode
    {attribute 'hide'}
	eMode:							E_RequestMode;						// Current mode
    {attribute 'hide'}
	eModePrevious:					E_RequestMode;						// Previous mode	
END_VAR

// https://github.com/PeterZerlauth/Tc3_Component

{attribute 'TcRpcEnable':='1'}
METHOD PUBLIC M_RequestMode : BOOL
VAR_INPUT
	eMode:		E_RequestMode;
END_VAR
IF THIS^.eMode = eMode THEN
	M_RequestMode:= TRUE;
ELSE
	eModeRequest:= eMode;	
END_IF
END_METHOD

{attribute 'TcRpcEnable':='1'}
METHOD PUBLIC M_RequestState : BOOL
VAR_INPUT
	eRequest:	E_RequestState;
END_VAR
// Request component states / Command Pattern
CASE eRequest OF
	E_RequestState.Undefined:
		M_RequestState:= TRUE;
		
	E_RequestState.Start:
		IF eState = E_State.Execute THEN
			M_RequestState:= TRUE;
		ELSE
			eStateRequest:= eRequest;				
		END_IF
		
	E_RequestState.Pause:
		IF eState >= E_State.Paused THEN
			M_RequestState:= TRUE;
		ELSE
			IF eStateRequest < eRequest THEN
				eStateRequest:= eRequest;				
			END_IF		
		END_IF
		
	E_RequestState.Hold:
		IF eState >= E_State.Held THEN
			M_RequestState:= TRUE;
		ELSE
			IF eStateRequest < eRequest THEN
				eStateRequest:= eRequest;				
			END_IF		
		END_IF
		
	E_RequestState.Complete:
		IF eState = E_State.Completed THEN
			M_RequestState:= TRUE;
		ELSE
			IF eStateRequest < eRequest THEN
				eStateRequest:= eRequest;				
			END_IF		
		END_IF
		
	E_RequestState.Stop:
		IF eState = E_State.Stopped THEN
			M_RequestState:= TRUE;
		ELSE
			IF eStateRequest < eRequest THEN
				eStateRequest:= eRequest;				
			END_IF		
		END_IF
		
	E_RequestState.Abort:
		IF eState = E_State.Aborted THEN
			M_RequestState:= TRUE;
		ELSE
			IF eStateRequest < eRequest THEN
				eStateRequest:= eRequest;				
			END_IF		
		END_IF

	E_RequestState.Reset:
		IF eState = E_State.Idle THEN
			M_RequestState:= TRUE;
		ELSE
			eStateRequest:= eRequest;			
		END_IF
END_CASE
END_METHOD

METHOD PROTECTED M_Aborted
VAR_INPUT
END_VAR
END_METHOD

METHOD PROTECTED M_Aborting : BOOL // Return state complete
VAR_INPUT
END_VAR
// State Aborting
M_Aborting:= TRUE;
END_METHOD

METHOD PROTECTED M_Completed
VAR_INPUT
END_VAR
END_METHOD

METHOD PROTECTED M_Completing : BOOL // Return state complete
VAR_INPUT
END_VAR
// State Completing
M_Completing:= True;
END_METHOD

METHOD PROTECTED M_Execute : BOOL // Return state complete
VAR_INPUT
END_VAR
M_Execute:= True;
END_METHOD

METHOD PROTECTED M_Held
VAR_INPUT
END_VAR
END_METHOD

METHOD PROTECTED M_Holding : BOOL // Return state complete
VAR_INPUT
END_VAR
// State Holding
M_Holding:= True;
END_METHOD

METHOD PROTECTED M_Idle
VAR_INPUT
END_VAR
// State Idle
END_METHOD

METHOD PROTECTED M_Initialise
VAR_INPUT
END_VAR
END_METHOD

METHOD PROTECTED M_Paused // Return state complete
VAR_INPUT
END_VAR
END_METHOD

METHOD PROTECTED M_Pausing : BOOL
VAR_INPUT
END_VAR
// State Holding
M_Pausing:= True;
END_METHOD

METHOD PROTECTED M_Resetting : BOOL // Return state complete
VAR_INPUT
END_VAR
// State Resetting
M_Resetting:= True;
END_METHOD

METHOD PROTECTED M_Resuming : BOOL // Return state complete
VAR_INPUT
END_VAR
// State Holding
M_Resuming:= True;
END_METHOD

METHOD PROTECTED M_Running
VAR_INPUT
END_VAR
// Will be called in all running states, for monitorings which not only in one state active
END_METHOD

METHOD PROTECTED M_Starting : BOOL // Return state complete
VAR_INPUT
END_VAR
// State Starting
M_Starting:= True;
END_METHOD

METHOD PROTECTED M_Stopped
VAR_INPUT
END_VAR
END_METHOD

METHOD PROTECTED M_Stopping : BOOL // Return state complete
VAR_INPUT
END_VAR
// State Stopping
M_Stopping:= True;
END_METHOD

METHOD PROTECTED M_Unholding : BOOL // Return state complete
VAR_INPUT
END_VAR
// State Holding
M_Unholding:= True;
END_METHOD

METHOD FB_init : BOOL
VAR_INPUT
	bInitRetains : BOOL; // if TRUE, the retain variables are initialized (warm start / cold start)
	bInCopyCode : BOOL:= TRUE;
END_VAR
M_Initialise();
END_METHOD

METHOD PUBLIC M_Cycle
VAR_INPUT
END_VAR
fbInfo();
fbEvent();
fbSequence();

// Handle Module Type Package states
CASE eState OF
	E_State.Undefined:
		M_Initialise();
		eMode:= E_RequestMode.Automatic;
		eState:= E_State.Idle;
				
	E_State.Resetting:
		M_Running();
		IF M_Resetting() THEN
			eState:= E_State.Idle;
			eStateRequest:= E_RequestState.Undefined;
			fbSequence.M_Reset();
		END_IF
		CASE eStateRequest OF
			E_RequestState.Stop:
				eState:= E_State.Stopping;
				fbSequence.M_Reset();
				
			E_RequestState.Abort:
				eState:= E_State.Aborting;
				fbSequence.M_Reset();
				fbSequence.M_Save();
				
		END_CASE
		
	E_State.Idle:
		M_Running();
		M_Idle();
		CASE eStateRequest OF
			
			E_RequestState.Start:
				eState:= E_State.Starting;
				fbSequence.M_Reset();
				
			E_RequestState.Stop:
				eState:= E_State.Stopping;
				fbSequence.M_Reset();
				
			E_RequestState.Abort:
				eState:= E_State.Aborting;
				fbSequence.M_Reset();
				fbSequence.M_Save();
				
			ELSE
				eStateRequest:= E_RequestState.Undefined;
				
		END_CASE

	E_State.Starting:
		M_Running();
		IF M_Starting() THEN
			eState:= E_State.Execute;
			eStateRequest:= E_RequestState.Undefined;
			fbSequence.M_Restore();

		END_IF
		CASE eStateRequest OF
			
			E_RequestState.Stop:
				eState:= E_State.Stopping;
				
			E_RequestState.Abort:
				eState:= E_State.Aborting;
				
		END_CASE

	E_State.Execute:
		M_Running();
		IF M_Execute() THEN
			CASE eStateRequest OF
				
				E_RequestState.Complete:
					eState:= E_State.Completing;
					fbSequence.M_Reset();
					
			END_CASE
		END_IF
		CASE eStateRequest OF
			E_RequestState.Complete:;
			E_RequestState.Stop:
				eState:= E_State.Stopping;
				fbSequence.M_Reset();
				
			E_RequestState.Abort:
				eState:= E_State.Aborting;
				fbSequence.M_Reset();

			E_RequestState.Hold:
				eState:= E_State.Holding;
				fbSequence.M_Reset();
				
			E_RequestState.Pause:
				eState:= E_State.Pausing;
				fbSequence.M_Reset();
				
			ELSE
				eStateRequest:= E_RequestState.Undefined;
				
		END_CASE
		fbSequence.M_Save();
		
	E_State.Stopping:
		M_Running();
		IF M_Stopping() THEN
			eState:= E_State.Stopped;
			eStateRequest:= E_RequestState.Undefined;
			fbSequence.M_Reset();
		END_IF
		CASE eStateRequest OF
			
			E_RequestState.Abort:
				eState:= E_State.Aborting;
				fbSequence.M_Reset();
				fbSequence.M_Save();
				
		END_CASE

	E_State.Stopped:
		M_Stopped();
		CASE eStateRequest OF
			
			E_RequestState.Abort:
				eState:= E_State.Aborting;
				fbSequence.M_Reset();
				fbSequence.M_Save();
				
			E_RequestState.Reset:
				eState:= E_State.Resetting;
				fbSequence.M_Reset();
				
		ELSE
			eStateRequest:= E_RequestState.Undefined;				
		END_CASE
		
		
	E_State.Aborting:
		IF M_Aborting() THEN
			eState:= E_State.Aborted;
			eStateRequest:= E_RequestState.Undefined;
			fbSequence.M_Reset();
			fbSequence.M_Save();
		END_IF
		
	E_State.Aborted:
		M_Aborted();
		CASE eStateRequest OF
			
			E_RequestState.Reset:
				eState:= E_State.Resetting;
				fbSequence.M_Reset();
				
		ELSE
			eStateRequest:= E_RequestState.Undefined;				
		END_CASE

		
	E_State.Pausing:
		M_Running();
		IF M_Pausing() THEN
			eState:= E_State.Paused;
			eStateRequest:= E_RequestState.Undefined;
			fbSequence.M_Reset();
		END_IF
		CASE eStateRequest OF
			
			E_RequestState.Stop:
				eState:= E_State.Stopping;
				fbSequence.M_Reset();
				
			E_RequestState.Abort:
				eState:= E_State.Aborting;
				fbSequence.M_Reset();
				fbSequence.M_Save();

		END_CASE
		
	
	E_State.Paused:
		M_Running();
		M_Paused();
		CASE eStateRequest OF
			
			E_RequestState.Start:
				eState:= E_State.Resuming;
				fbSequence.M_Reset();
				
			E_RequestState.Stop:
				eState:= E_State.Stopping;
				fbSequence.M_Reset();
				
			E_RequestState.Abort:
				eState:= E_State.Aborting;
				fbSequence.M_Reset();
				fbSequence.M_Save();
						
		ELSE
			eStateRequest:= E_RequestState.Undefined;

		END_CASE
		
	E_State.Resuming:
		M_Running();
		IF M_Resuming() THEN
			eState:= E_State.Execute;
			fbSequence.M_Reset();
		END_IF
		CASE eStateRequest OF
			
			E_RequestState.Stop:
				eState:= E_State.Stopping;
				fbSequence.M_Reset();
				
			E_RequestState.Abort:
				eState:= E_State.Aborting;
				fbSequence.M_Reset();
				fbSequence.M_Save();
				
		END_CASE

	E_State.Holding:
		M_Running();
		IF M_Holding() THEN
			eState:= E_State.Held;
			eStateRequest:= E_RequestState.Undefined;
			fbSequence.M_Reset();
		END_IF
		CASE eStateRequest OF
			
			E_RequestState.Stop:
				eState:= E_State.Stopping;
				fbSequence.M_Reset();
				
			E_RequestState.Abort:
				eState:= E_State.Aborting;
				fbSequence.M_Reset();
				fbSequence.M_Save();

		END_CASE

	E_State.Held:
		M_Running();
		M_Held();
		CASE eStateRequest OF
			
			E_RequestState.Start:
				eState:= E_State.Unholding;
				fbSequence.M_Reset();

			E_RequestState.Stop:
				eState:= E_State.Stopping;
				fbSequence.M_Reset();
				
			E_RequestState.Abort:
				eState:= E_State.Aborting;
				fbSequence.M_Reset();
				fbSequence.M_Save();
				
			ELSE
				eStateRequest:= E_RequestState.Undefined;

		END_CASE
		
	E_State.Unholding:
		M_Running();
		IF M_Unholding() THEN
			eState:= E_State.Execute;
			fbSequence.M_Reset();
		END_IF
		CASE eStateRequest OF
			
			E_RequestState.Stop:
				eState:= E_State.Stopping;
				fbSequence.M_Reset();
				
			E_RequestState.Abort:
				eState:= E_State.Aborting;
				fbSequence.M_Reset();			
				fbSequence.M_Save();		

		END_CASE
		
	E_State.Completing:
		M_Running();
		IF M_Completing() THEN
			eState:= E_State.Completed;
			eStateRequest:= E_RequestState.Undefined;
			fbSequence.M_Reset();
		END_IF
		CASE eStateRequest OF
			
			E_RequestState.Stop:
				eState:= E_State.Stopping;
				fbSequence.M_Reset();
				
			E_RequestState.Abort:
				eState:= E_State.Aborting;
				fbSequence.M_Reset();
				fbSequence.M_Save();
		END_CASE
		
	E_State.Completed:
		M_Running();
		M_Completed();
		CASE eStateRequest OF
			
			E_RequestState.Stop:
				eState:= E_State.Stopping;
				fbSequence.M_Reset();
				
			E_RequestState.Abort:
				eState:= E_State.Aborting;
				fbSequence.M_Reset();
					
			E_RequestState.Reset:
				eState:= E_State.Resetting;
				fbSequence.M_Reset();
				fbSequence.M_Save();
				
			ELSE
				eStateRequest:= E_RequestState.Undefined;
				
		END_CASE
		
END_CASE

IF eModeRequest <> E_RequestMode.Undefined THEN
	IF eMode <> eModeRequest THEN
		eModePrevious:= eMode;
		eMode:= eModeRequest;
		M_OnMode(eMode, eModePrevious);
	END_IF
END_IF
eModeRequest:= E_RequestMode.Undefined;
	
// Detect state changed
IF eStatePrevious <> eState THEN
	M_OnState(eState, eStatePrevious);
	eStatePrevious:= eState;
END_IF
END_METHOD

METHOD PUBLIC M_Notify
VAR_INPUT
	iSender:		I_Component;
	eRequest:		E_RequestState;
END_VAR
M_RequestState(eRequest);

// Notify all other components in observer
fbEvent.P_Observer.M_Notify(iSender, eRequest);
END_METHOD

METHOD PROTECTED M_OnMode
VAR_INPUT
	eMode:							E_RequestMode;						// Current mode
	eModePrevious:					E_RequestMode;						// Previous mode	
END_VAR
END_METHOD

METHOD Protected M_OnState
VAR_INPUT
	eState:							E_State;						// Current state
	eStatePrevious:					E_State;						// Previous state	
END_VAR
END_METHOD

PROPERTY PUBLIC P_Event : I_Event
GET
P_Event:= fbEvent;
END_GET
END_PROPERTY

{attribute 'OPC.UA.DA.Property' := '1'}
{attribute 'monitoring' := 'call'}
PROPERTY PUBLIC P_Info : I_Info
GET
P_Info:= fbInfo;
END_GET
END_PROPERTY

{attribute 'OPC.UA.DA.Property' := '1'}
{attribute 'monitoring' := 'call'}
PROPERTY PUBLIC P_Mode : E_RequestMode
GET
P_Mode:= eMode;
END_GET
END_PROPERTY

{attribute 'OPC.UA.DA.Property' := '1'}
{attribute 'monitoring' := 'call'}
PROPERTY PUBLIC P_Sequence : I_Sequence
GET
P_Sequence:= fbSequence;
END_GET
END_PROPERTY

{attribute 'OPC.UA.DA.Property' := '1'}
{attribute 'monitoring' := 'call'}
PROPERTY PUBLIC P_State : E_State
GET
P_State:= eState;
END_GET
END_PROPERTY

END_FUNCTION_BLOCK

// Object/FB_Object
FUNCTION_BLOCK FB_Object IMPLEMENTS I_Object
VAR_INPUT
END_VAR
VAR_OUTPUT
END_VAR
VAR
END_VAR

END_FUNCTION_BLOCK

// Function/FB_Function
FUNCTION_BLOCK FB_Function EXTENDS FB_Component
VAR_INPUT
END_VAR
VAR_OUTPUT
END_VAR
VAR
END_VAR

END_FUNCTION_BLOCK

// Layers/Layer/FB_Layer
FUNCTION_BLOCK FB_Layer EXTENDS FB_Component IMPLEMENTS I_Layer
VAR_INPUT
END_VAR
VAR_OUTPUT
END_VAR
VAR
	tDelay:				TIME;
	tTimeout:			TIME;
	iNext:				I_Component;	// Chain of Responsibility behavioral design pattern 
	fbList:				FB_ListComponent;
END_VAR

METHOD PUBLIC M_Attach
VAR_INPUT
	iComponent:		I_Component;
END_VAR
fbList.M_Add(iComponent);
iComponent.P_Event.P_Observer.M_Attach(THIS^);
fbEvent.P_Observer.M_Attach(iComponent);
END_METHOD

METHOD PUBLIC M_Dettach
VAR_INPUT
	iComponent:		I_Component;
END_VAR
fbList.M_Remove(iComponent);
iComponent.P_Event.P_Observer.M_Detach(THIS^);
fbEvent.P_Observer.M_Detach(iComponent);
END_METHOD

METHOD M_Notify
VAR_INPUT
	iSender:		I_Component;
	eRequest:		E_RequestState;
END_VAR
SUPER^.M_Notify(iSender, eRequest);
IF iNext <> 0 THEN
	iNext.M_Notify(iSender, eRequest);
END_IF
END_METHOD

METHOD PROTECTED M_Resetting : BOOL (* Return state complete*)
VAR
	nIndex: 		DINT;
END_VAR
M_Resetting:= TRUE;
WHILE nIndex < fbList.P_Length DO
	IF fbList.M_Index(nIndex).M_RequestState(E_RequestState.Reset) THEN
		;
	ELSE
		M_Resetting:= FALSE;
	END_IF	
	nIndex:= nIndex + 1; 
END_WHILE
END_METHOD

METHOD PROTECTED M_Starting : BOOL (* Return state complete*)
VAR
	nIndex: 		DINT;
END_VAR
M_Starting:= TRUE;
WHILE nIndex < fbList.P_Length DO
	IF fbList.M_Index(nIndex).M_RequestState(E_RequestState.Start) THEN
		;
	ELSE
		M_Starting:= FALSE;
	END_IF	
	nIndex:= nIndex + 1; 
END_WHILE
END_METHOD

{attribute 'OPC.UA.DA.Property' := '1'}
{attribute 'monitoring' := 'call'}
PROPERTY PUBLIC P_Delay : TIME
GET
P_Delay:= tDelay;
END_GET
SET
tDelay:= P_Delay;
END_SET
END_PROPERTY

{attribute 'OPC.UA.DA.Property' := '1'}
{attribute 'monitoring' := 'call'}
PROPERTY P_List : I_ListComponent
GET
P_List:= fbList;
END_GET
END_PROPERTY

{attribute 'OPC.UA.DA.Property' := '1'}
{attribute 'monitoring' := 'call'}
PROPERTY PUBLIC P_Next : I_Component
GET
P_Next:= iNext;
END_GET
SET
iNext:= P_Next;
END_SET
END_PROPERTY

{attribute 'OPC.UA.DA.Property' := '1'}
{attribute 'monitoring' := 'call'}
PROPERTY PUBLIC P_Timeout : TIME
GET
P_Timeout:= tTimeout;
END_GET
SET
tTimeout:= P_Timeout;
END_SET
END_PROPERTY

END_FUNCTION_BLOCK

// Layers/Layer/I_Layer
INTERFACE I_Layer EXTENDS I_Component

METHOD PUBLIC M_Attach
VAR_INPUT
	iComponent:		I_Component;
END_VAR
END_METHOD

METHOD PUBLIC M_Dettach
VAR_INPUT
	iComponent:		I_Component;
END_VAR
END_METHOD

{attribute 'OPC.UA.DA.Property' := '1'}
{attribute 'monitoring' := 'call'}
PROPERTY PUBLIC P_Delay : TIME
GET
END_GET
SET
END_SET
END_PROPERTY

{attribute 'OPC.UA.DA.Property' := '1'}
{attribute 'monitoring' := 'call'}
PROPERTY P_List : I_ListComponent
GET
END_GET
END_PROPERTY

{attribute 'OPC.UA.DA.Property' := '1'}
{attribute 'monitoring' := 'call'}
PROPERTY PUBLIC P_Next : I_Component
GET
END_GET
SET
END_SET
END_PROPERTY

{attribute 'OPC.UA.DA.Property' := '1'}
{attribute 'monitoring' := 'call'}
PROPERTY PUBLIC P_Timeout : TIME
GET
END_GET
SET
END_SET
END_PROPERTY

END_INTERFACE

// List/I_ListComponent
INTERFACE I_ListComponent Extends I_ListBase

METHOD PUBLIC M_Add : BOOL
VAR_INPUT
	iObject: 	I_Component;
END_VAR
END_METHOD

METHOD PUBLIC M_Find : DINT
VAR_INPUT
	iObject: 	I_Component;
END_VAR
END_METHOD

METHOD PUBLIC M_Index : I_Component
VAR_INPUT
	Index: 	DINT;
END_VAR
END_METHOD

METHOD PUBLIC M_Remove : BOOL
VAR_INPUT
	iObject: 	I_Component;
END_VAR
END_METHOD

END_INTERFACE

// List/FB_ListComponent
{attribute 'no_explicit_call' := 'do not call this POU directly'} 
FUNCTION_BLOCK FB_ListComponent IMPLEMENTS I_ListComponent
VAR
	nLength:		DINT;
	pList: 			POINTER TO I_Component;
	{IF (defined (release))}
    	{attribute 'hide'}
	{END_IF}
	aList:			POINTER TO POINTER TO ARRAY [0..Parameters.nList] OF I_Component:=ADR(pList);
END_VAR

// https://github.com/PeterZerlauth/Tc3_Component

METHOD FB_exit : BOOL
VAR_INPUT
	bInCopyCode : BOOL; // if TRUE, the exit method is called for exiting an instance that is copied afterwards (online change).
END_VAR
M_Clear();
END_METHOD

METHOD PUBLIC M_Add : BOOL
VAR_INPUT
	iObject: 	I_Component;
END_VAR
VAR
	pOldList: 	POINTER TO I_Component;
END_VAR
IF iObject <> 0 THEN
	// First Item
	IF pList = 0 THEN
		nLength:= nLength + 1;
		pList:= __NEW(POINTER TO I_Component,DINT_TO_UDINT(nLength));
	ELSE
		// Item already in List
		IF M_Find(iObject) = -1 THEN
			// backup 
			pOldList:= pList;
			// new Length
			nLength:= nLength + 1;
			// new pointer
			pList:= __NEW(POINTER TO I_Component,DINT_TO_UDINT(nLength));
			// restore
			Memcpy(pList,pOldList, SIZEOF(POINTER TO I_Component)*DINT_TO_UDINT(nLength -1));
			// delete old
			__DELETE(pOldList);
		ELSE
			M_Add:= FALSE;	
			RETURN;
		END_IF
	END_IF
	IF pList = 0 THEN
		RETURN;
	END_IF
	// add new Object
	pList[nLength-1]:= iObject;
	M_Add:= TRUE;
ELSE
	M_Add:= FALSE;	
END_IF
END_METHOD

METHOD PUBLIC M_Clear : BOOL
// Clear
IF pList <> 0 THEN
	nLength:= 0;
	__DELETE(pList);
END_IF
M_Clear:= TRUE;
END_METHOD

METHOD PUBLIC M_Find : DINT
VAR_INPUT
	iObject: 	I_Component;
END_VAR
VAR
	nIndex: 	UINT;
END_VAR
// Find
M_Find := -1;
WHILE nIndex < nLength DO
    IF (pList[nIndex] = iObject) THEN
        M_Find := nIndex;
        RETURN;
    END_IF
	nIndex := nIndex + 1;
END_WHILE
END_METHOD

METHOD PUBLIC M_Index : I_Component
VAR_INPUT
	Index: 	DINT;
END_VAR
// Index
IF Index <= nLength THEN
	M_Index:= pList[Index];
END_IF
END_METHOD

METHOD PUBLIC M_Remove : BOOL
VAR_INPUT
	iObject: 	I_Component;
END_VAR
VAR
	pOldList:			POINTER TO I_Component;
	nPosition: 			DINT;
END_VAR
// Remove
IF iObject <> 0 THEN
	// First Item
	IF nLength >= 0 THEN
		// Item already in List
		nPosition:= M_Find(iObject);
		IF nPosition <> -1 THEN
			// backup 
			pOldList:= pList;
			// new Length
			nLength:= nLength -1;
			// new pointer
			pList:= __NEW(POINTER TO I_Component,DINT_TO_UDINT(nLength));
			// restore lower part
			Memcpy(pList,pOldList, SIZEOF(POINTER TO I_Object) * DINT_TO_UDINT(nPosition));
			//pList[nPosition]:= iObject;
			Memcpy(pList + (SIZEOF(POINTER TO I_Component)*nPosition),pOldList + (SIZEOF(POINTER TO I_Component)*(nPosition + 1)), SIZEOF(POINTER TO I_Component) * DINT_TO_UDINT(nLength - nPosition));
			// delete old
			__DELETE(pOldList);
		ELSE
			M_Remove:= FALSE;	
			RETURN;
		END_IF
	ELSE
		M_Remove:= FALSE;	
		RETURN;
	END_IF
	M_Remove:= TRUE;
ELSE
	M_Remove:= FALSE;	
END_IF
END_METHOD

{attribute 'OPC.UA.DA.Property' := '1'}
{attribute 'monitoring' := 'call'}
PROPERTY PUBLIC P_Length : DINT
GET
P_Length:= nLength;
END_GET
END_PROPERTY

END_FUNCTION_BLOCK

// Layers/FB_Layers
FUNCTION_BLOCK FB_Layers IMPLEMENTS I_Cycle, I_Layers
VAR_INPUT
	fbE0:							FB_Layer;
	fbE1:							FB_Layer;
	fbOn:							FB_Layer;
END_VAR
VAR_OUTPUT
END_VAR
VAR
END_VAR

METHOD M_Cycle
fbE0.M_Cycle();
fbE1.M_Cycle();
fbOn.M_Cycle();
END_METHOD

{attribute 'OPC.UA.DA.Property' := '1'}
{attribute 'monitoring' := 'call'}
PROPERTY PUBLIC P_E0 : I_Layer
GET
P_E0:= fbE0;
END_GET
END_PROPERTY

{attribute 'OPC.UA.DA.Property' := '1'}
{attribute 'monitoring' := 'call'}
PROPERTY PUBLIC P_E1 : I_Layer
GET
P_E1:= fbE1;
END_GET
END_PROPERTY

{attribute 'OPC.UA.DA.Property' := '1'}
{attribute 'monitoring' := 'call'}
PROPERTY PUBLIC P_On : I_Layer
GET
P_On:= fbOn;
END_GET
END_PROPERTY

END_FUNCTION_BLOCK

// Layers/I_Layers
INTERFACE I_Layers EXTENDS I_Object

{attribute 'OPC.UA.DA.Property' := '1'}
{attribute 'monitoring' := 'call'}
PROPERTY PUBLIC P_E0 : I_Layer
GET
END_GET
END_PROPERTY

{attribute 'OPC.UA.DA.Property' := '1'}
{attribute 'monitoring' := 'call'}
PROPERTY PUBLIC P_E1 : I_Layer
GET
END_GET
END_PROPERTY

{attribute 'OPC.UA.DA.Property' := '1'}
{attribute 'monitoring' := 'call'}
PROPERTY PUBLIC P_On : I_Layer
GET
END_GET
END_PROPERTY

END_INTERFACE

// List/FB_ListObject
{attribute 'no_explicit_call' := 'do not call this POU directly'} 
FUNCTION_BLOCK FB_ListObject IMPLEMENTS I_ListObject
VAR
	nLength:		DINT;
	pList: 			POINTER TO I_Object;
	{IF (defined (release))}
    	{attribute 'hide'}
	{END_IF}
	aList:			POINTER TO POINTER TO ARRAY [0..Parameters.nList] OF I_Object:=ADR(pList);
END_VAR

// https://github.com/PeterZerlauth/Tc3_Component

METHOD FB_exit : BOOL
VAR_INPUT
	bInCopyCode : BOOL; // if TRUE, the exit method is called for exiting an instance that is copied afterwards (online change).
END_VAR
M_Clear();
END_METHOD

METHOD PUBLIC M_Add : BOOL
VAR_INPUT
	Object: 	I_Object;
END_VAR
VAR
	pOldList: 	POINTER TO I_Object;
END_VAR
IF Object <> 0 THEN
	// First Item
	IF pList = 0 THEN
		nLength:= nLength + 1;
		pList:= __NEW(POINTER TO I_Object,DINT_TO_UDINT(nLength));
	ELSE
		// Item already in List
		IF M_Find(Object) = -1 THEN
			// backup 
			pOldList:= pList;
			// new Length
			nLength:= nLength + 1;
			// new pointer
			pList:= __NEW(POINTER TO I_Object,DINT_TO_UDINT(nLength));
			// restore
			Memcpy(pList,pOldList, SIZEOF(POINTER TO I_Object)*DINT_TO_UDINT(nLength -1));
			// delete old
			__DELETE(pOldList);
		ELSE
			M_Add:= FALSE;	
			RETURN;
		END_IF
	END_IF
	IF pList = 0 THEN
		RETURN;
	END_IF
	// add new Object
	pList[nLength-1]:= Object;
	M_Add:= TRUE;
ELSE
	M_Add:= FALSE;	
END_IF
END_METHOD

METHOD PUBLIC M_Clear : bool
IF pList <> 0 THEN
	nLength:= 0;
	__DELETE(pList);
END_IF
M_Clear:= True;
END_METHOD

METHOD PUBLIC M_Find : DINT
VAR_INPUT
	Object: 	I_Object;
END_VAR
VAR
	nIndex: 	UINT;
END_VAR
// Object already in List
M_Find := -1;
WHILE nIndex < nLength DO
    IF (pList[nIndex] = Object) THEN
        M_Find := nIndex;
        RETURN;
    END_IF
	nIndex := nIndex + 1;
END_WHILE
END_METHOD

METHOD PUBLIC M_Index : I_Object
VAR_INPUT
	Index: 	DINT;
END_VAR
IF Index <= nLength THEN
	M_Index:= pList[Index];
END_IF
END_METHOD

METHOD PUBLIC M_Remove : BOOL
VAR_INPUT
	Object: 	I_Object;
END_VAR
VAR
	pOldList:			POINTER TO I_Object;
	nPosition: 			DINT;
END_VAR
IF Object <> 0 THEN
	// First Item
	IF nLength >= 0 THEN
		// Item already in List
		nPosition:= M_Find(Object);
		IF nPosition <> -1 THEN
			// backup 
			pOldList:= pList;
			// new Length
			nLength:= nLength -1;
			// new pointer
			pList:= __NEW(POINTER TO I_Object,DINT_TO_UDINT(nLength));
			// restore lower part
			Memcpy(pList,pOldList, SIZEOF(POINTER TO I_Object) * DINT_TO_UDINT(nPosition));
			//pList[nPosition]:= iObject;
			Memcpy(pList + (SIZEOF(POINTER TO I_Object)*nPosition),pOldList + (SIZEOF(POINTER TO I_Object)*(nPosition + 1)), SIZEOF(POINTER TO I_Object) * DINT_TO_UDINT(nLength - nPosition));
			// delete old
			__DELETE(pOldList);
		ELSE
			M_Remove:= FALSE;	
			RETURN;
		END_IF
	ELSE
		M_Remove:= FALSE;	
		RETURN;
	END_IF
	M_Remove:= TRUE;
ELSE
	M_Remove:= FALSE;	
END_IF
END_METHOD

{attribute 'OPC.UA.DA.Property' := '1'}
{attribute 'monitoring' := 'call'}
PROPERTY PUBLIC P_Length : DINT
GET
P_Length:= nLength;
END_GET
END_PROPERTY

END_FUNCTION_BLOCK

// List/I_ListObject
INTERFACE I_ListObject Extends I_ListBase

METHOD PUBLIC M_Add : BOOL
VAR_INPUT
	Object: 	I_Object;
END_VAR
END_METHOD

METHOD PUBLIC M_Find : DINT
VAR_INPUT
	Object: 	I_Object;
END_VAR
END_METHOD

METHOD PUBLIC M_Index : I_Object
VAR_INPUT
	Index: 	DINT;
END_VAR
END_METHOD

METHOD PUBLIC M_Remove : BOOL
VAR_INPUT
	Object: 	I_Object;
END_VAR
END_METHOD

END_INTERFACE

// Logger/FB_AbstractLogger
FUNCTION_BLOCK ABSTRACT FB_AbstractLogger IMPLEMENTS I_Logger
VAR
	eLogLevel:					E_Event:= E_Event.Verbose;		// Log level for the logger
END_VAR

// https://github.com/PeterZerlauth/Tc3_Component
// Abstract Logger as base for all loggers

METHOD PUBLIC M_Log
VAR_INPUT
	{attribute 'analysis' := '-33'}
	stEvent	: ST_Event;
END_VAR
END_METHOD

PROPERTY PUBLIC P_LogLevel : E_Event
GET
P_LogLevel:= eLogLevel;
END_GET
SET
eLogLevel:= P_LogLevel;
END_SET
END_PROPERTY

END_FUNCTION_BLOCK

// Logger/FB_GlobalLogger
FUNCTION_BLOCK FB_GlobalLogger EXTENDS FB_AbstractLogger
VAR 
    {attribute 'hide'}
	aEvent:						ARRAY [0..nSize - 1] OF ST_Event;
END_VAR
VAR CONSTANT 
	nSize: DINT:= 50; 
END_VAR

// https://github.com/PeterZerlauth/Tc3_Component

METHOD PUBLIC M_Find : DINT
VAR_INPUT
	stEvent:	ST_Event;
END_VAR
VAR 
	nIndex:		DINT;
END_VAR
// Find event in buffer
M_Find := -1;

WHILE nIndex < nSize - 1 DO
	IF (aEvent[nIndex].iSource = stEvent.iSource) AND_THEN
    	(aEvent[nIndex].eEventType = stEvent.eEventType) AND_THEN
		(aEvent[nIndex].sInstance = stEvent.sInstance) AND_THEN
		(aEvent[nIndex].sClass = stEvent.sClass) AND_THEN
		(aEvent[nIndex].sMessage = stEvent.sMessage) THEN
        M_Find := nIndex;
        RETURN;
    END_IF
	nIndex := nIndex + 1;
END_WHILE
END_METHOD

METHOD public M_Log
VAR_INPUT
	{attribute 'analysis' := '-33'}
	stEvent	: ST_Event;
END_VAR
VAR
	nIndex:				DINT;
	sMessage:			STRING(255);
END_VAR
IF (nIndex:=  M_Find(stEvent)) >= 0 THEN
	;
ELSE
	IF stEvent.eEventType >= SUPER^.eLogLevel THEN
		MEMCPY(ADR(aEvent[1]), ADR(aEvent[0]), DINT_TO_UDINT(SIZEOF(ST_Event) * (nSize - 1)));
		aEvent[0]:= stEvent;
		sMessage:= Concat(Concat(stEvent.sInstance, ' | fbObserver.P_Length = 0 | '), stEvent.sDefault);
		CASE stEvent.eEventType OF
			E_Event.Error:
				ADSLOGSTR( msgCtrlMask := ADSLOG_MSGTYPE_ERROR , msgFmtStr := '%s', strArg := sMessage);
			E_Event.Warning:
				ADSLOGSTR( msgCtrlMask := ADSLOG_MSGTYPE_WARN , msgFmtStr := '%s', strArg := sMessage);
			E_Event.Information:
				ADSLOGSTR( msgCtrlMask := ADSLOG_MSGTYPE_HINT , msgFmtStr := '%s', strArg := sMessage);
			E_Event.Debug:
				ADSLOGSTR( msgCtrlMask := ADSLOG_MSGTYPE_HINT, msgFmtStr := '%s', strArg := sMessage);
			E_Event.Verbose:
				ADSLOGSTR( msgCtrlMask := ADSLOG_MSGTYPE_HINT , msgFmtStr := '%s', strArg := sMessage);
		END_CASE
	END_IF
END_IF
END_METHOD

END_FUNCTION_BLOCK

// Logger/FB_ListObject_1
{attribute 'no_explicit_call' := 'do not call this POU directly'} 
FUNCTION_BLOCK FB_ListObject_1 IMPLEMENTS I_ListObject
VAR
	nLength:		DINT;
	pList: 			POINTER TO I_Object;
	{IF (defined (release))}
    	{attribute 'hide'}
	{END_IF}
	aList:			POINTER TO POINTER TO ARRAY [0..Parameters.nList] OF I_Object:=ADR(pList);
END_VAR

// https://github.com/PeterZerlauth/Tc3_Component

METHOD FB_exit : BOOL
VAR_INPUT
	bInCopyCode : BOOL; // if TRUE, the exit method is called for exiting an instance that is copied afterwards (online change).
END_VAR
M_Clear();
END_METHOD

METHOD PUBLIC M_Add : BOOL
VAR_INPUT
	Object: 	I_Object;
END_VAR
VAR
	pOldList: 	POINTER TO I_Object;
END_VAR
IF Object <> 0 THEN
	// First Item
	IF pList = 0 THEN
		nLength:= nLength + 1;
		pList:= __NEW(POINTER TO I_Object,DINT_TO_UDINT(nLength));
	ELSE
		// Item already in List
		IF M_Find(Object) = -1 THEN
			// backup 
			pOldList:= pList;
			// new Length
			nLength:= nLength + 1;
			// new pointer
			pList:= __NEW(POINTER TO I_Object,DINT_TO_UDINT(nLength));
			// restore
			Memcpy(pList,pOldList, SIZEOF(POINTER TO I_Object)*DINT_TO_UDINT(nLength -1));
			// delete old
			__DELETE(pOldList);
		ELSE
			M_Add:= FALSE;	
			RETURN;
		END_IF
	END_IF
	IF pList = 0 THEN
		RETURN;
	END_IF
	// add new Object
	pList[nLength-1]:= Object;
	M_Add:= TRUE;
ELSE
	M_Add:= FALSE;	
END_IF
END_METHOD

METHOD PUBLIC M_Clear : bool
IF pList <> 0 THEN
	nLength:= 0;
	__DELETE(pList);
END_IF
M_Clear:= True;
END_METHOD

METHOD PUBLIC M_Find : DINT
VAR_INPUT
	Object: 	I_Object;
END_VAR
VAR
	nIndex: 	UINT;
END_VAR
// Object already in List
M_Find := -1;
WHILE nIndex < nLength DO
    IF (pList[nIndex] = Object) THEN
        M_Find := nIndex;
        RETURN;
    END_IF
	nIndex := nIndex + 1;
END_WHILE
END_METHOD

METHOD PUBLIC M_Index : I_Object
VAR_INPUT
	Index: 	DINT;
END_VAR
IF Index <= nLength THEN
	M_Index:= pList[Index];
END_IF
END_METHOD

METHOD PUBLIC M_Remove : BOOL
VAR_INPUT
	Object: 	I_Object;
END_VAR
VAR
	pOldList:			POINTER TO I_Object;
	nPosition: 			DINT;
END_VAR
IF Object <> 0 THEN
	// First Item
	IF nLength >= 0 THEN
		// Item already in List
		nPosition:= M_Find(Object);
		IF nPosition <> -1 THEN
			// backup 
			pOldList:= pList;
			// new Length
			nLength:= nLength -1;
			// new pointer
			pList:= __NEW(POINTER TO I_Object,DINT_TO_UDINT(nLength));
			// restore lower part
			Memcpy(pList,pOldList, SIZEOF(POINTER TO I_Object) * DINT_TO_UDINT(nPosition));
			//pList[nPosition]:= iObject;
			Memcpy(pList + (SIZEOF(POINTER TO I_Object)*nPosition),pOldList + (SIZEOF(POINTER TO I_Object)*(nPosition + 1)), SIZEOF(POINTER TO I_Object) * DINT_TO_UDINT(nLength - nPosition));
			// delete old
			__DELETE(pOldList);
		ELSE
			M_Remove:= FALSE;	
			RETURN;
		END_IF
	ELSE
		M_Remove:= FALSE;	
		RETURN;
	END_IF
	M_Remove:= TRUE;
ELSE
	M_Remove:= FALSE;	
END_IF
END_METHOD

{attribute 'OPC.UA.DA.Property' := '1'}
{attribute 'monitoring' := 'call'}
PROPERTY PUBLIC P_Length : DINT
GET
P_Length:= nLength;
END_GET
END_PROPERTY

END_FUNCTION_BLOCK

// Logger/FB_Logger
FUNCTION_BLOCK FB_Logger EXTENDS FB_AbstractLogger
VAR
    {attribute 'hide'}
	nLength:					DINT;
    {attribute 'hide'}
	aEvent:						ARRAY [0..nSize - 1] OF ST_Event;
    {attribute 'hide'}
	nIndex: 					DINT;
    {attribute 'hide'}
	nTimestamp: 				ULINT;
END_VAR	
VAR CONSTANT 
	nSize: DINT:= 50; 
END_VAR

// https://github.com/PeterZerlauth/Tc3_Component
// Execute each secound
IF nTimestamp < F_GetSystemTime() THEN
	nTimestamp:= F_GetSystemTime() + 10000000;
	nIndex:= 0;
	WHILE nIndex < nLength DO
		IF aEvent[nIndex].stFlags.bActive THEN
			IF aEvent[nIndex].stFlags.bRemove THEN
				aEvent[nIndex].stFlags.bActive:= FALSE;
			END_IF
		ELSE
			M_Delete(nIndex);
		END_IF
		nIndex := nIndex + 1;
	END_WHILE
END_IF

METHOD PUBLIC M_Delete : BOOL
VAR_INPUT
	nIndex: 			DINT;
END_VAR
// new Length
nLength:= nLength -1;
//pList[nPosition]:= iObject;
Memcpy(ADR(aEvent[nIndex]), ADR(aEvent[nIndex +1]), SIZEOF(POINTER TO ST_Event) * DINT_TO_UDINT(nSize - nIndex));
END_METHOD

METHOD PUBLIC M_Find : DINT
VAR_INPUT
	stEvent:	ST_Event;
END_VAR
VAR 
	nIndex:		DINT;
END_VAR
// Find event in buffer
M_Find := -1;
WHILE nIndex < nLength DO
	IF (aEvent[nIndex].iSource = stEvent.iSource) AND_THEN
    	(aEvent[nIndex].eEventType = stEvent.eEventType) AND_THEN
		(aEvent[nIndex].sInstance = stEvent.sInstance) AND_THEN
		(aEvent[nIndex].sClass = stEvent.sClass) AND_THEN
		(aEvent[nIndex].sMessage = stEvent.sMessage) THEN
        M_Find := nIndex;
        RETURN;
    END_IF
	nIndex := nIndex + 1;
END_WHILE
END_METHOD

METHOD PUBLIC M_Log
VAR_INPUT
	stEvent:		ST_Event;
END_VAR
VAR
	nIndex:			DINT;
END_VAR
IF (nIndex:=  M_Find(stEvent)) >= 0 THEN
	// Update existing events
	aEvent[nIndex].sArguments:= stEvent.sArguments;
	aEvent[nIndex].sDefault:= stEvent.sDefault;
	aEvent[nIndex].stFlags:= stEvent.stFlags;
ELSE
	// add new event
	aEvent[nLength]:= stEvent;
	nLength:= nLength + 1;
END_IF
END_METHOD

METHOD PUBLIC M_Reset
VAR_INPUT
END_VAR
// Reset all events
nLength:= 0;
Memset(ADR(aEvent), 0, SIZEOF(aEvent));
END_METHOD

{attribute 'OPC.UA.DA.Property' := '1'}
{attribute 'monitoring' := 'call'}
{attribute 'suppress_wrn_C0410'}
PROPERTY PUBLIC P_Events : REFERENCE TO ARRAY [0..nSize - 1] OF ST_Event
GET
P_Events REF= aEvent;
END_GET
SET
P_Events REF= aEvent;
END_SET
END_PROPERTY

{attribute 'OPC.UA.DA.Property' := '1'}
{attribute 'monitoring' := 'call'}
PROPERTY PUBLIC P_Length : DINT
GET
P_Length:= nLength;
END_GET
END_PROPERTY

END_FUNCTION_BLOCK

// Logger/FB_TcLogger
FUNCTION_BLOCK FB_TcLogger EXTENDS FB_AbstractLogger
VAR 
	aEvent:						ARRAY [0..nSize - 1] OF ST_Event;
END_VAR
VAR CONSTANT 
	nSize: DINT:= 50; 
END_VAR

// https://github.com/PeterZerlauth/Tc3_Component

METHOD PUBLIC M_Find : DINT
VAR_INPUT
	stEvent:	ST_Event;
END_VAR
VAR 
	nIndex:		DINT;
END_VAR
// Find event in buffer
M_Find := -1;
WHILE nIndex < nSize - 1 DO
	IF (aEvent[nIndex].iSource = stEvent.iSource) AND_THEN
    	(aEvent[nIndex].eEventType = stEvent.eEventType) AND_THEN
		(aEvent[nIndex].sInstance = stEvent.sInstance) AND_THEN
		(aEvent[nIndex].sClass = stEvent.sClass) AND_THEN
		(aEvent[nIndex].sMessage = stEvent.sMessage) THEN
        M_Find := nIndex;
        RETURN;
    END_IF
	nIndex := nIndex + 1;
END_WHILE
END_METHOD

METHOD M_Log
VAR_INPUT
	{attribute 'analysis' := '-33'}
	stEvent	: ST_Event;
END_VAR
VAR
	nIndex:				DINT;
	sMessage:			STRING(255);
END_VAR
IF (nIndex:=  M_Find(stEvent)) >= 0 THEN
	;
ELSE
	IF stEvent.eEventType >= SUPER^.eLogLevel THEN
		MEMCPY(ADR(aEvent[1]), ADR(aEvent[0]), DINT_TO_UDINT(SIZEOF(ST_Event) * (nSize - 1)));
		aEvent[0]:= stEvent;
		sMessage:= Concat(Concat(stEvent.sInstance, ' | '), stEvent.sDefault);
		CASE stEvent.eEventType OF
			E_Event.Error:
				ADSLOGSTR( msgCtrlMask := ADSLOG_MSGTYPE_ERROR , msgFmtStr := '%s', strArg := sMessage);
			E_Event.Warning:
				ADSLOGSTR( msgCtrlMask := ADSLOG_MSGTYPE_WARN , msgFmtStr := '%s', strArg := sMessage);
			E_Event.Information:
				ADSLOGSTR( msgCtrlMask := ADSLOG_MSGTYPE_HINT , msgFmtStr := '%s', strArg := sMessage);
			E_Event.Debug:
				ADSLOGSTR( msgCtrlMask := ADSLOG_MSGTYPE_HINT, msgFmtStr := '%s', strArg := sMessage);
			E_Event.Verbose:
				ADSLOGSTR( msgCtrlMask := ADSLOG_MSGTYPE_HINT , msgFmtStr := '%s', strArg := sMessage);
		END_CASE
	END_IF
END_IF
END_METHOD

METHOD PUBLIC M_Reset
VAR_INPUT
END_VAR
// Reset all events
Memset(ADR(aEvent), 0, SIZEOF(aEvent));
END_METHOD

END_FUNCTION_BLOCK

// Module/FB_Module
FUNCTION_BLOCK FB_Module EXTENDS FB_Component IMPLEMENTS I_Module
VAR_INPUT
END_VAR
VAR_OUTPUT
END_VAR
VAR
	fbLayers:					FB_Layers;
	fbFunctions:				FB_Layer;
	fbLogger:					FB_Logger;
	fbTcLogger:					FB_TcLogger;
END_VAR

// https://github.com/PeterZerlauth/Tc3_Component

METHOD PROTECTED M_Aborted
VAR_INPUT
END_VAR
SUPER^.M_Aborted();
fbEvent.M_AddSTRING(P_Info.P_ID);
fbEvent.M_Info('Module %s aborted, reset', 2);
END_METHOD

METHOD PROTECTED M_Completing : BOOL // Return state complete
VAR_INPUT
END_VAR

VAR
	nIndex: INT;
END_VAR
M_Completing:= TRUE;
WHILE nIndex < fbFunctions.P_List.P_Length DO
	CASE fbFunctions.P_List.M_Index(nIndex).P_State OF
		E_State.Idle,E_State.Completed,E_State.Stopped,E_State.Aborted:
			;
		ELSE
			M_Completing:= FALSE;
	END_CASE
	nIndex:= nIndex +1;
END_WHILE
END_METHOD

METHOD PUBLIC M_Cycle
VAR_INPUT
END_VAR
SUPER^.M_Cycle();


fbLayers.M_Cycle();

fbFunctions.M_Cycle();

fbLogger();
fbTcLogger();
END_METHOD

METHOD PROTECTED M_Holding : BOOL // Return state complete
VAR_INPUT
END_VAR

VAR
	nIndex: INT;
END_VAR
M_Holding:= TRUE;
WHILE nIndex < fbFunctions.P_List.P_Length DO
	CASE fbFunctions.P_List.M_Index(nIndex).P_State OF
		E_State.Idle,E_State.Completed,E_State.Stopped,E_State.Aborted:
			;
		ELSE
			M_Holding:= FALSE;
	END_CASE
	nIndex:= nIndex +1;
END_WHILE
END_METHOD

METHOD PROTECTED M_Idle
VAR_INPUT
END_VAR
SUPER^.M_Idle();
fbEvent.M_AddSTRING(P_Info.P_ID);
fbEvent.M_Info('Module %s not started', 3);
END_METHOD

METHOD PROTECTED M_Initialise
VAR_INPUT
END_VAR

VAR
	fbLoggerFactory: INT;
END_VAR
SUPER^.M_Initialise();

fbLayers.fbE0.P_Next:= fbLayers.fbE1;
fbLayers.fbE1.P_Next:= fbLayers.fbOn;
fbLayers.fbOn.P_Next:= THIS^;
END_METHOD

METHOD PROTECTED M_OnMode
VAR_INPUT
	eMode:							E_RequestMode;						// Current mode
	eModePrevious:					E_RequestMode;						// Previous mode	
END_VAR
CASE eMode OF
	E_RequestMode.Semiauto, E_RequestMode.Automatic:
		IF eModePrevious = E_RequestMode.Manual THEN
			fbEvent.M_AddSTRING(TO_STRING(eModePrevious));
			fbEvent.M_AddSTRING(TO_STRING(eMode));
			fbEvent.M_Abort('Mode changed form %s to %s', 4);
		END_IF
	E_RequestMode.Manual:
		fbEvent.M_AddSTRING(TO_STRING(eModePrevious));
		fbEvent.M_AddSTRING(TO_STRING(eMode));
		fbEvent.M_Debug('Mode changed form %s to %s');
END_CASE
END_METHOD

METHOD PROTECTED M_Pausing : BOOL
VAR_INPUT
END_VAR

VAR
	nIndex: INT;
END_VAR
M_Pausing:= TRUE;
WHILE nIndex < fbFunctions.P_List.P_Length DO
	CASE fbFunctions.P_List.M_Index(nIndex).P_State OF
		E_State.Idle,E_State.Completed,E_State.Stopped,E_State.Aborted:
			;
		ELSE
			M_Pausing:= FALSE;
	END_CASE
	nIndex:= nIndex +1;
END_WHILE
END_METHOD

METHOD PROTECTED M_Resetting : BOOL
VAR_INPUT
END_VAR
M_Resetting:= SUPER^.M_Resetting();
fbLayers.fbE0.M_RequestState(E_RequestState.Reset);
fbLayers.fbE1.M_RequestState(E_RequestState.Reset);
fbLayers.fbOn.M_RequestState(E_RequestState.Reset);
fbFunctions.M_RequestState(E_RequestState.Reset);
fbLogger.M_Reset();
fbTcLogger.M_Reset();
END_METHOD

METHOD PROTECTED M_Resuming : BOOL // Return state complete
VAR_INPUT
END_VAR
IF fbLayers.fbE0.M_RequestState(E_RequestState.Start) THEN
	M_Resuming:= TRUE;
	fbLogger.M_Reset();
	fbTcLogger.M_Reset();
END_IF
END_METHOD

METHOD PROTECTED M_Running
VAR_INPUT
END_VAR
END_METHOD

METHOD PROTECTED M_Starting : BOOL
VAR_INPUT
END_VAR
VAR
	bReturn:			BOOL;
END_VAR
CASE fbSequence.P_Number OF
	E_Sequence.Start:
		bReturn:= fbLayers.fbE0.M_RequestState(E_RequestState.Start);
		fbSequence.M_Await('Start layer 0', T#5S, T#1S, FALSE, bReturn, 10);
		
	10:
		bReturn:= fbLayers.fbE1.M_RequestState(E_RequestState.Start);
		fbSequence.M_Await('Start layer 1', T#5S, T#1S, FALSE, bReturn, 20);
		
	20:
		bReturn:= fbLayers.fbOn.M_RequestState(E_RequestState.Start);
		fbSequence.M_Await('Start layer 1', T#5S, T#1S, FALSE, bReturn, E_Sequence.Done);
		
	E_Sequence.Done:
		M_Starting:= TRUE;
END_CASE
END_METHOD

METHOD PROTECTED M_Stopped
VAR_INPUT
END_VAR
SUPER^.M_Stopped();
fbEvent.M_AddSTRING(P_Info.P_ID);
fbEvent.M_Info('Module %s stopped, reset', 5);
END_METHOD

METHOD PROTECTED M_Unholding : BOOL // Return state complete
VAR_INPUT
END_VAR
IF fbLayers.fbE0.M_RequestState(E_RequestState.Start) THEN
	M_Unholding:= TRUE;
	fbLogger.M_Reset();
	fbTcLogger.M_Reset();
END_IF
END_METHOD

{attribute 'OPC.UA.DA.Property' := '1'}
{attribute 'monitoring' := 'call'}
{attribute 'suppress_wrn_C0410'}
PROPERTY PUBLIC P_Layers : I_Layers
GET
P_Layers:= fbLayers;
END_GET
END_PROPERTY

END_FUNCTION_BLOCK

// Module/I_Module
INTERFACE I_Module EXTENDS I_Component

{attribute 'OPC.UA.DA.Property' := '1'}
{attribute 'monitoring' := 'call'}
{attribute 'suppress_wrn_C0410'}
PROPERTY PUBLIC P_Layers : I_Layers
GET
END_GET
END_PROPERTY

END_INTERFACE

// Utils/Analog/AnalogInput
{attribute 'reflection'} 
FUNCTION_BLOCK AnalogInput IMPLEMENTS I_AnalogChannel
VAR_INPUT
END_VAR
VAR_OUTPUT
END_VAR
VAR
	sIdentifier:				STRING(25);	// Equipment ID
	Channel						AT%I*: INT;	// Link to input
END_VAR

// https://github.com/PeterZerlauth/Tc3_Component

PROPERTY PUBLIC P_ID : String(25)
GET
P_ID:= sIdentifier;
END_GET
END_PROPERTY

PROPERTY P_State : EPlcMappingStatus
GET
P_State:= F_GetMappingStatus(ADR(Channel), SIZEOF(INT));
END_GET
END_PROPERTY

PROPERTY PUBLIC P_Value : Lreal
GET
P_Value:= INT_TO_LREAL(Channel);
END_GET
SET
PUBLIC 
VAR
END_VAR
Channel:= LREAL_TO_INT(P_Value);
END_SET
END_PROPERTY

END_FUNCTION_BLOCK

// Utils/Analog/I_AnalogChannel
INTERFACE I_AnalogChannel EXTENDS I_Channel

PROPERTY P_Value : LREAL
GET
END_GET
SET
END_SET
END_PROPERTY

END_INTERFACE

// Utils/Digital/I_Channel
INTERFACE I_Channel EXTENDS I_Object

PROPERTY PUBLIC P_ID : String(25)
GET
END_GET
END_PROPERTY

PROPERTY P_State : EPlcMappingStatus
GET
END_GET
END_PROPERTY

END_INTERFACE

// Utils/Analog/AnalogInputREAL
{attribute 'reflection'} 
FUNCTION_BLOCK AnalogInputREAL IMPLEMENTS I_AnalogChannel
VAR_INPUT
END_VAR
VAR_OUTPUT
END_VAR
VAR
	sIdentifier:				STRING(25);	// Equipment ID
	Channel			AT%I*: REAL;	// Link to input
END_VAR

// https://github.com/PeterZerlauth/Tc3_Component

PROPERTY PUBLIC P_ID : String(25)
GET
P_ID:= sIdentifier;
END_GET
END_PROPERTY

PROPERTY P_State : EPlcMappingStatus
GET
P_State:= F_GetMappingStatus(ADR(Channel), SIZEOF(INT));
END_GET
END_PROPERTY

PROPERTY PUBLIC P_Value : Lreal
GET
P_Value:= Channel;
END_GET
SET
PUBLIC 
VAR
END_VAR
Channel:= LREAL_TO_INT(P_Value);
END_SET
END_PROPERTY

END_FUNCTION_BLOCK

// Utils/Analog/AnalogOutput
{attribute 'reflection'} 
FUNCTION_BLOCK AnalogOutput IMPLEMENTS I_AnalogChannel
VAR_INPUT
END_VAR
VAR_OUTPUT
END_VAR
VAR
	sIdentifier:				STRING(25);	// Equipment ID
	Channel			AT%Q*: INT;	// Link to input
END_VAR

// https://github.com/PeterZerlauth/Tc3_Component

METHOD FB_init : BOOL
VAR_INPUT
	bInitRetains : BOOL; // if TRUE, the retain variables are initialized (warm start / cold start)
	bInCopyCode : BOOL;  // if TRUE, the instance afterwards gets moved into the copy code (online change)
	ID:				STRING(25);
END_VAR
THIS^.sIdentifier:= ID;
END_METHOD

PROPERTY PUBLIC P_ID : String(25)
GET
P_ID:= sIdentifier;
END_GET
END_PROPERTY

PROPERTY P_State : EPlcMappingStatus
GET
P_State:= F_GetMappingStatus(ADR(Channel), SIZEOF(INT));
END_GET
END_PROPERTY

PROPERTY PUBLIC P_Value : Lreal
GET
P_Value:= INT_TO_LREAL(Channel);
END_GET
SET
PUBLIC 
VAR
END_VAR
Channel:= LREAL_TO_INT(P_Value);
END_SET
END_PROPERTY

END_FUNCTION_BLOCK

// Utils/Digital/FB_DigitalInput
{attribute 'reflection'} 
FUNCTION_BLOCK FB_DigitalInput IMPLEMENTS I_DigitalChannel
VAR_INPUT
	tDebounce:			TIME:= T#50MS;
END_VAR
VAR_OUTPUT
END_VAR
VAR

	sIdentifier:				STRING(25);	// Equipment ID
	bChannel				AT%I*: BOOL;	// Link to input
	fbDebounce:				FB_Debounce;
END_VAR

// https://github.com/PeterZerlauth/Tc3_Component
fbDebounce(bInput:= bChannel, tTime:= tDebounce);

PROPERTY PUBLIC P_ID : String(25)
GET
P_ID:= sIdentifier;
END_GET
END_PROPERTY

PROPERTY P_State : EPlcMappingStatus
GET
P_State:= F_GetMappingStatus(ADR(bChannel), SIZEOF(BOOL));
END_GET
END_PROPERTY

PROPERTY PUBLIC P_Value : bool
GET
P_Value:= fbDebounce.bValue;
END_GET
SET
PUBLIC 
VAR
END_VAR
END_SET
END_PROPERTY

END_FUNCTION_BLOCK

// Utils/Digital/I_DigitalChannel
INTERFACE I_DigitalChannel EXTENDS I_Channel

PROPERTY P_Value : bool
GET
END_GET
SET
END_SET
END_PROPERTY

END_INTERFACE

// Utils/FB_Debounce
FUNCTION_BLOCK FB_Debounce 
VAR_INPUT
	bInput:				BOOL;
	tTime:				TIME;
END_VAR
VAR_OUTPUT
	bValue:				BOOL;
END_VAR
VAR
	fbTimerOn:			Ton;
	fbTimerOff:			Ton;
END_VAR

// https://github.com/PeterZerlauth/Tc3_Component
IF bInput THEN
	fbTimerOn(IN:= TRUE, PT:= tTime);
	fbTimerOff(IN:= FALSE);
	IF fbTimerOn.Q THEN
		bValue:= TRUE;
	END_IF
ELSE
	fbTimerOff(IN:= TRUE, PT:= tTime);
	fbTimerOn(IN:= FALSE);
	IF fbTimerOff.Q THEN
		bValue:= FALSE;
	END_IF	
END_IF

PROPERTY PUBLIC P_Value : BOOL
GET
P_Value:= bValue;
END_GET
END_PROPERTY

END_FUNCTION_BLOCK

// Utils/Digital/FB_DigitalOutput
{attribute 'reflection'} 
FUNCTION_BLOCK FB_DigitalOutput IMPLEMENTS I_DigitalChannel
VAR_INPUT
END_VAR
VAR_OUTPUT
END_VAR
VAR
	sIdentifier:				STRING(25);		// Equipment ID
	Channel			AT%Q*: BOOL;	// Link to output
END_VAR

// https://github.com/PeterZerlauth/Tc3_Component

PROPERTY PUBLIC P_ID : STRING(25)
GET
P_ID:= sIdentifier;
END_GET
END_PROPERTY

PROPERTY P_State : EPlcMappingStatus
GET
P_State:= F_GetMappingStatus(adr(Channel), sizeof(BOOL));
END_GET
END_PROPERTY

PROPERTY PUBLIC P_Value : bool
GET
P_Value:= Channel;
END_GET
SET
PUBLIC 
VAR
END_VAR
Channel:= P_Value;
END_SET
END_PROPERTY

END_FUNCTION_BLOCK

// Utils/File/FB_File
{attribute 'no_explicit_call'} 
FUNCTION_BLOCK FB_File
VAR
    fbCreateDir:	FB_CreateDir;
	fbOpen:			FB_FileOpen;
	fbRead:			FB_FileRead;
	fbLoad:			FB_FileLoad;
	fbWrite:		FB_FileWrite;
	fbClose:		FB_FileClose;
	fbDelete:		FB_FileDelete;
END_VAR
VAR_OUTPUT
	nError:			UDINT;
END_VAR

// https://github.com/PeterZerlauth/Tc3_Component
fbCreateDir();
fbLoad();
fbOpen();
fbClose();
fbDelete();
fbWrite();
fbRead();

METHOD PUBLIC M_Append : BOOL
VAR_INPUT
	Text:			STRING(255);
END_VAR
IF fbWrite.bExecute THEN
	IF fbWrite.bError THEN
		nError:= fbWrite.nErrId;
		fbWrite.bExecute:= FALSE;
	ELSIF fbWrite.bBusy THEN
		;
	ELSE
		M_Append:= TRUE;
		fbWrite.bExecute:= FALSE;
	END_IF
ELSE
	fbWrite.bExecute:= TRUE;
	fbWrite.pWriteBuff:= ADR(Text);
	fbWrite.cbWriteLen:= INT_TO_UDINT(Len(Text));
END_IF
END_METHOD

METHOD PUBLIC M_AppendLine : BOOL
VAR_INPUT
	Text:			STRING(255);
END_VAR
Text:= Concat(Text, '$R');
M_AppendLine:= M_Append(Text);
END_METHOD

METHOD PUBLIC M_Close : BOOL
VAR_INPUT
END_VAR
IF fbClose.bExecute THEN
	IF fbClose.hFile = 0 THEN
		fbClose.bExecute:= FALSE;
		M_Close:= TRUE;
	ELSIF fbClose.bError THEN
		fbClose.bExecute:= FALSE;
		nError:= fbClose.nErrId;
	ELSIF fbClose.bBusy THEN
		;
	ELSE
		nError:= 0;	
		fbRead.hFile:= 0;
		fbWrite.hFile:= 0;
		fbClose.hFile:= 0;
		fbClose.bExecute:= FALSE;
		M_Close:= TRUE;
	END_IF
ELSE
	fbClose.bExecute:= TRUE;
END_IF
END_METHOD

METHOD PUBLIC M_Create : BOOL
VAR_INPUT
	PathName:		STRING(255);
END_VAR
VAR
	nTemp: INT;
END_VAR
VAR_INST
	nPosition: INT;
END_VAR
nTemp := FIND(RIGHT(PathName, LEN(PathName) - nPosition), '\');
if nTemp <> 0 then
	IF fbCreateDir.bExecute THEN
		IF NOT fbCreateDir.bBusy THEN
			nPosition := nPosition + nTemp;
			fbCreateDir.bExecute:= FALSE;
		END_IF
	ELSE
		fbCreateDir.bExecute:= TRUE;
		fbCreateDir.ePath:= PATH_GENERIC;
		fbCreateDir.sPathName:= Left(PathName, nPosition + nTemp);
	END_IF
ELSE
	IF M_Open(PathName) THEN
		M_Create:= TRUE;
		nPosition:= 0;
	END_IF
END_IF
END_METHOD

METHOD PUBLIC M_Delete : BOOL
VAR_INPUT
	PathName:		STRING(255);
END_VAR
IF fbDelete.bExecute THEN
	IF fbDelete.bError THEN
		fbDelete.bExecute:= FALSE;
		M_Delete:= TRUE;
	ELSIF fbDelete.bBusy THEN
		;
	ELSE
		fbDelete.bExecute:= FALSE;
		M_Delete:= TRUE;
	END_IF
ELSE
	fbDelete.bExecute:= TRUE;
	fbDelete.sPathName:= PathName;
	fbDelete.ePath:= E_OpenPath.PATH_GENERIC;
END_IF
END_METHOD

METHOD PUBLIC M_Load : BOOL
VAR_INPUT
	PathName:		STRING(255);
	Value:			ANY;
END_VAR
IF fbLoad.bExecute THEN
	IF fbLoad.bError THEN
		nError:= fbLoad.nErrId;
		fbLoad.bExecute:= FALSE;
	ELSIF fbLoad.bBusy THEN
		;
	ELSE
		M_Load:= TRUE;
	END_IF
ELSE
	fbLoad.sPathName:= PathName;
	fbLoad.bExecute:= TRUE;
	fbLoad.pReadBuff:= Value.pValue;
	fbLoad.cbReadLen:= DINT_TO_UDINT(Value.diSize);
END_IF
END_METHOD

METHOD PUBLIC M_Open : BOOL
VAR_INPUT
	PathName:		STRING(255);
END_VAR
IF fbOpen.bExecute THEN
	IF fbOpen.bError THEN
		nError:= fbOpen.nErrId;
		fbOpen.bExecute:= FALSE;
	ELSIF fbOpen.bBusy THEN
		;
	ELSE
		fbRead.hFile:= fbOpen.hFile;
		fbWrite.hFile:= fbOpen.hFile;
		fbClose.hFile:= fbOpen.hFile;
		fbOpen.bExecute:= FALSE;
		M_Open:= TRUE;
	END_IF	
ELSE
	fbOpen.bExecute:= TRUE;
	fbOpen.sPathName:= PathName;
	fbOpen.nMode:= (FOPEN_MODEAPPEND OR FOPEN_MODEPLUS OR FOPEN_MODETEXT);
END_IF
END_METHOD

METHOD PUBLIC M_Read : BOOL
VAR_INPUT
	Value:		ANY;
END_VAR
IF fbRead.bExecute THEN
	IF fbRead.bError THEN
		nError:= fbRead.nErrId;
		fbRead.bExecute:= FALSE;
	ELSIF fbRead.bBusy THEN
		;
	ELSE
		fbRead.bExecute:= FALSE;
		M_Read:= TRUE;
	END_IF
ELSE
	fbRead.bExecute:= TRUE;
	fbRead.pReadBuff:= Value.pValue;
	fbRead.cbReadLen:= DINT_TO_UDINT(Value.diSize);
END_IF
END_METHOD

METHOD PUBLIC M_Write : BOOL
VAR_INPUT
	Value:		ANY;
END_VAR
IF fbWrite.bExecute THEN
	IF fbWrite.bError THEN
		nError:= fbWrite.nErrId;
		fbWrite.bExecute:= FALSE;
	ELSIF fbWrite.bBusy THEN
		M_Write:= FALSE;
	ELSE
		M_Write:= TRUE;
		fbWrite.bExecute:= FALSE;
	END_IF
ELSE
	fbWrite.bExecute:= TRUE;
	fbRead.pReadBuff:= Value.pValue;
	fbRead.cbReadLen:= DINT_TO_UDINT(Value.diSize);
END_IF
END_METHOD

PROPERTY PUBLIC P_Error : UDINT
GET
P_Error:= nError;
END_GET
END_PROPERTY

END_FUNCTION_BLOCK

// Utils/File/I_File
INTERFACE I_File

METHOD PUBLIC M_Append : BOOL
VAR_INPUT
	sText:			STRING(255);
END_VAR
END_METHOD

METHOD PUBLIC M_AppendLine : BOOL
VAR_INPUT
	sText:			STRING(255);
END_VAR
END_METHOD

METHOD PUBLIC M_Close : BOOL
VAR_INPUT
END_VAR
END_METHOD

METHOD PUBLIC M_Create : BOOL
VAR_INPUT
	sPathName:		T_MaxString;
END_VAR
END_METHOD

METHOD PUBLIC M_Delete : BOOL
VAR_INPUT
	sPathName:		T_MaxString;
END_VAR
END_METHOD

METHOD PUBLIC M_Load : BOOL
VAR_INPUT
	sPathName:		T_MaxString;
	pData:			PVOID;
	nData:			UDINT;
END_VAR
END_METHOD

METHOD PUBLIC M_Open : BOOL
VAR_INPUT
	sPathName:		T_MaxString;
END_VAR
END_METHOD

METHOD PUBLIC M_Read : BOOL
VAR_INPUT
	Value:		ANY;
END_VAR
END_METHOD

METHOD PUBLIC M_Write : BOOL
VAR_INPUT
	Value:		ANY;
END_VAR
END_METHOD

PROPERTY PUBLIC P_Error : UDINT
GET
END_GET
END_PROPERTY

END_INTERFACE

// Utils/FB_ArrayDint
FUNCTION_BLOCK FB_ArrayDint VAR_GENERIC CONSTANT nLength: DINT:= 1; END_VAR
VAR_INPUT
END_VAR
VAR_OUTPUT
END_VAR
VAR
	nValues:			ARRAY [0..nLength - 1] OF DINT;
END_VAR

END_FUNCTION_BLOCK
